REGION Network 10: J no magnet pallet ///Empty pallet full
   RUNG wire#powerrail
      Contact( "AlwaysTRUE" )
      Contact( "Station_Sys".Auto.Mode )
      wire#w1
      I_Contact( "AutoProcessControl".J_MagnetLine.Robot2PickPrimit )
      I_Contact( "iJ-magnetLiftingPalletDischargeDetection" )
      Coil( "ST10_TipDB".Global."6"[4] )
   END_RUNG
   RUNG wire#w1
      Contact( "iJ-magnetTakeShaftDetection" )
      { S7_Templates := "time_type := Time" } "TON".TON[48].TON(pt := T#3S, et =>)
      Coil( "ST10_TipDB".Global."6"[5] )
   END_RUNG
   // the same network as SCL:
   #_w1 := "AlwaysTRUE" AND "Station_Sys".Auto.Mode;
   "ST10_TipDB".Global."6"[4] := #_w1 AND NOT "AutoProcessControl".J_MagnetLine.Robot2PickPrimit AND NOT "iJ-magnetLiftingPalletDischargeDetection";
   "TON".TON[48].TON(IN := #_w1 AND "iJ-magnetTakeShaftDetection", PT := T#3S);
   "ST10_TipDB".Global."6"[5] := "TON".TON[48].Q;
END_REGION

REGION Network 11: K no magnet pallet ///Empty pallet full
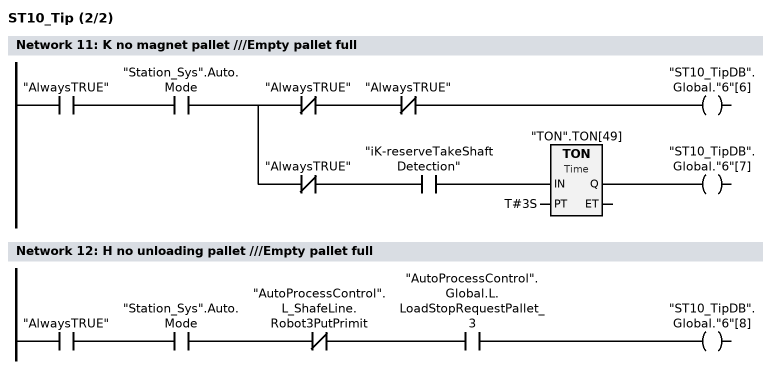
   RUNG wire#powerrail
      Contact( "AlwaysTRUE" )
      Contact( "Station_Sys".Auto.Mode )
      wire#w1
      I_Contact( "AlwaysTRUE" )
      I_Contact( "AlwaysTRUE" )
      Coil( "ST10_TipDB".Global."6"[6] )
   END_RUNG
   RUNG wire#w1
      I_Contact( "AlwaysTRUE" )
      Contact( "iK-reserveTakeShaftDetection" )
      { S7_Templates := "time_type := Time" } "TON".TON[49].TON(pt := T#3S, et =>)
      Coil( "ST10_TipDB".Global."6"[7] )
   END_RUNG
   // the same network as SCL:
   #_w1 := "AlwaysTRUE" AND "Station_Sys".Auto.Mode;
   "ST10_TipDB".Global."6"[6] := #_w1 AND NOT "AlwaysTRUE" AND NOT "AlwaysTRUE";
   "TON".TON[49].TON(IN := #_w1 AND NOT "AlwaysTRUE" AND "iK-reserveTakeShaftDetection", PT := T#3S);
   "ST10_TipDB".Global."6"[7] := "TON".TON[49].Q;
END_REGION

REGION Network 12: H no unloading pallet ///Empty pallet full
   RUNG wire#powerrail
      Contact( "AlwaysTRUE" )
      Contact( "Station_Sys".Auto.Mode )
      I_Contact( "AutoProcessControl".L_ShafeLine.Robot3PutPrimit )
      Contact( "AutoProcessControl".Global.L.LoadStopRequestPallet_3 )
      Coil( "ST10_TipDB".Global."6"[8] )
   END_RUNG
   // the same network as SCL:
   "ST10_TipDB".Global."6"[8] := "AlwaysTRUE" AND "Station_Sys".Auto.Mode AND NOT "AutoProcessControl".L_ShafeLine.Robot3PutPrimit AND "AutoProcessControl".Global.L.LoadStopRequestPallet_3;
END_REGION
END_FUNCTION

FUNCTION "CylinderCtrl_V2" : Void   // FC3011, SCL
TITLE = CylinderV3
{ S7_Optimized_Access := 'FALSE' }
AUTHOR : JM
FAMILY : RCS
VERSION : 18.2
// this function is only used for cylinder control
// stored: AutoNumber false, SetENOAutomatically true
   VAR_INPUT
      iReset : Bool;   // reset action
      iRun : Bool;   // system run
      iEStop : Bool;   // e_stop monitor
      iManualMode : Bool;   // manual mode
      iAutoMode : Bool;   // auto mode
      iEnableAlarm : Bool;   // alarm will popup up
      iPulse100mS : Bool;   // pulse *100ms
      iPulse1S : Bool;   // pulse*1s
      iCyDBNO : Word;   // Interface data block number
      iCyCounts : Int;   // total counts of cylinder to be used[must be>=1 and <=100]
      iDevAlarmDBNum : Word;   // Device Alarm DataBlock Alarm
   END_VAR
   VAR_TEMP
      CyInterface : "Cyl";
      CyRany : Any;
      cyRSany AT CyRany : Struct
         SyntaxID : Byte;
         DataType : Byte;
         RepetitionFactor : Int;
         DB_Number : Word;
         MemoryAreaAddress : DWord;
      END_STRUCT;
      CyDany : Any;
      CyDSany AT CyDany : Struct
         SyntaxID : Byte;
         DataType : Byte;
         RepetitionFactor : Int;
         DB_Number : Word;
         MemoryAreaAddress : DWord;
      END_STRUCT;
      tpCounts : Int;
      tpi : Int;
      tpRetVal : Int;
   END_VAR
BEGIN
   //---------------------------------------------------------------//
   //FunctionName:CylinderV3
   //FunctionDescription:Cylinder Control block
   //---------------------------------------------------------------//
   (*in:

   #iReset  Bool            reset action
   #iRun    Bool            system run
   #iE_stop Bool            e_stop monitor
   #iManualMode Bool        manual mode
   #iAutoMode   Bool        auto mode
   #iEnableAlarm    Bool        alarm will popup up
   #iPulse_100mS    Bool        pulse *100ms
   iPulse_1S   Bool        pulse*1s
   iCyDBNO Int Int     Interface data block number
   iCyCounts   Int     total counts OF "Cylinder" TO be used[must be>=1 AND <=100]

   //inout:
   //out:
   *)
   //---------------------------------------------------------------//
   //Version:V3
   //D&T:2016-11-14
   //Group:RCS
   //Author:JiangMing
   //-------------------------Modify1----------------------------------//
   //Version:
   //D&T:2016-11-17
   //Group: RCS
   //Author:JiangMing
   //Modify:Update cylinder no as output interface
   //-------------------------Modify2----------------------------------//
   //Version:       V18.3
   //D&T:           2020-06-11
   //Group:         RCS
   //Author:        JM
   //Modify:        1.MaxCylinder count 200 
   //               2.Refine alarm interface
   IF #iCyCounts > 200 THEN
       #tpCounts := 200;
   ELSE
       #tpCounts := #iCyCounts;
   END_IF;
   //input

   FOR #tpi := 0 TO #tpCounts-1 DO
       //****************************************************************************************//
       #cyRSany.SyntaxID := 16#10;
       #cyRSany.DataType := 16#02;
       #cyRSany.RepetitionFactor := 22;
       #cyRSany.DB_Number := #iCyDBNO;
       #cyRSany.MemoryAreaAddress := 16#8400_0000 OR (SHL(IN := INT_TO_DWORD(#tpi * 22), N := 3));///
       //-----------------------------//
       #CyDSany.SyntaxID := 16#10;
       #CyDSany.DataType := 16#02;
       #CyDSany.RepetitionFactor := 22;
       #CyDSany.DB_Number := 0;
       #CyDSany.MemoryAreaAddress := 16#8700_0000 OR (SHL(IN := INT_TO_DWORD(0), N := 3));///
       #tpRetVal := BLKMOV(SRCBLK := #CyRany, DSTBLK => #CyDany);
       //***************************************************************************************//
       "CylinderModule_V2"(iReset := #iReset,
                        iRun := #iRun,
                        iEStop := #iEStop,
                        iManualMode := #iManualMode,
                        iAutoMode := #iAutoMode,
                        iEnableAlarm := #iEnableAlarm,
                        iPulse100mS := #iPulse100mS,
                        iPulse1S := #iPulse1S,
                        iError := #CyInterface.In.Error,
                        iGoWorkInterlock := #CyInterface.In.GoWorkInterlock,
                        iGoHomeInterlock := #CyInterface.In.GoHomeInterlock,
                        iWorkPositionSensor := #CyInterface.In.WorkPositionSensor,
                        iHomePositionSensor := #CyInterface.In.HomePositionSensor,
                        iValveType := #CyInterface.In.ValveType,
                        iManualOutputType := #CyInterface.In.ManualOutputType,
                        iFaultTime := #CyInterface.In.FaultTime,
                        iOnPositionTime := #CyInterface.In.OnPositionTime,
                           ioResetOut:=#CyInterface.Inout.ResetOut,
                        ioGoWorkPosition := #CyInterface.Out.GoWorkPosition,
                        ioGoHomePosition := #CyInterface.Out.GoHomePosition,
                        oGoWP_ButtonActive => #CyInterface.Out.GoWPButtonActive,
                        oGoHP_ButtonActive => #CyInterface.Out.GoHPButtonActive,
                        ioGoWorkFault := #CyInterface.Out.GoWorkFault,
                        ioGoHomeFault := #CyInterface.Out.GoHomeFault,
                        ioSensorPositionFault := #CyInterface.Out.SensorPositionFault,
                        oCyNo => #CyInterface.Out.CyNO,
                        ioManualGoWork := #CyInterface.Inout.ManualGoWork,
                        ioManualGoHome := #CyInterface.Inout.ManualGoHome,
                        ioAutoGoWork := #CyInterface.Inout.AutoGoWork,
                        ioAutoGoHome := #CyInterface.Inout.AutoGoHome,
                        ioGoWorkTime := #CyInterface.S.GoWorkTime,
                        ioGoHomeTime := #CyInterface.S.GoHomeTime,
                        ioWorkFaultTime := #CyInterface.S.WorkFaultTime,
                        ioHomeFaultTime := #CyInterface.S.HomeFaultTime,
                        ioBothSensorOnTime := #CyInterface.S.BothSensorOnTime,
                        ioPulse100mSP := #CyInterface.S.Pulse100mSP,
                        ioAutoGoWorkP := #CyInterface.S.AutoGoWorkP,
                        ioAutoGoHomeP := #CyInterface.S.AutoGoHomeP,
                        ioGoWork100mSP := #CyInterface.S.GoWork100mSP,
                        ioGoHome100mSP := #CyInterface.S.GoHome100mSP,
                        ioBothSensorOn100mSP := #CyInterface.S.BothSensorOn100mSP,
                        ioAlarm := #CyInterface.S.Alarm,
                        ioSpare1 := #CyInterface.S.spare1,
                        ioSpare2 := #CyInterface.S.spare2);
       //*******************************************************************************//
         POKE_BOOL(area := 16#84,
                   bitOffset := 4 * (#tpi MOD 2) + 0,
                   byteOffset :=  #tpi / 2,
                   dbNumber := #iDevAlarmDBNum,
                   value := #CyInterface.Out.GoWorkFault);
         POKE_BOOL(area := 16#84,
                   bitOffset := 4 * (#tpi MOD 2) + 1,
                   byteOffset :=  #tpi / 2,
                   dbNumber := #iDevAlarmDBNum,
                   value := #CyInterface.Out.GoHomeFault);
         POKE_BOOL(area := 16#84,
                   bitOffset := 4 * (#tpi MOD 2) + 2,
                   byteOffset :=  #tpi / 2,
                   dbNumber := #iDevAlarmDBNum,
                   value := #CyInterface.Out.SensorPositionFault);
       #CyInterface.Out.CyNO := INT_TO_BYTE(#tpi+1);
       //output
       #cyRSany.SyntaxID := 16#10;
       #cyRSany.DataType := 16#02;
       #cyRSany.RepetitionFactor := 16;
       #cyRSany.DB_Number := 0;
       #cyRSany.MemoryAreaAddress := 16#8700_0000 OR (SHL(IN := INT_TO_DWORD(6), N := 3));///
       //-----------------------------//
       #CyDSany.SyntaxID := 16#10;
       #CyDSany.DataType := 16#02;
       #CyDSany.RepetitionFactor := 16;
       #CyDSany.DB_Number := #iCyDBNO;
       #CyDSany.MemoryAreaAddress := 16#8400_0000 OR (SHL(IN := INT_TO_DWORD(#tpi* 22 + 6), N := 3));///
       #tpRetVal := BLKMOV(SRCBLK := #CyRany, DSTBLK => #CyDany);
       //******************************************************************************//


   END_FOR;
END_FUNCTION

FUNCTION "ST10Cyl_interface1-10" : Void   // FC1020, LAD
{ S7_Optimized_Access := 'FALSE' }
// stored: AutoNumber false, SetENOAutomatically false
   VAR_INPUT
      AlwaysON : Bool;
      E_stop : Bool;
   END_VAR
   VAR_TEMP
      tTest : Bool;
      i : Int;
   END_VAR
BEGIN

REGION Network 1 (SCL): Cylinder 1-10 IO Interface (SCL)
   IF "Station_Sys".Manual.Mode THEN

       FOR #i := 1 TO 100 BY 1

       DO
           "ST10Cylinder".Cy[#i].In.ManualOutputType := TRUE;

       END_FOR;

   END_IF;

   //Cylinder1 IO  A-Loading-01HorizontalCylinder
   //Input
   "ST10Cylinder".Cy[1].In.WorkPositionSensor := "iA-Loading-01HorizontalCylinderInWP";
   "ST10Cylinder".Cy[1].In.HomePositionSensor := "iA-Loading-01HorizontalCylinderInHP";
   //Output
   "oA-Loading-01HorizontalCylinderToWP" := "ST10Cylinder".Cy[1].Out.GoWorkPosition;
   "oA-Loading-01HorizontalCylinderToHP" := "ST10Cylinder".Cy[1].Out.GoHomePosition;

   //Cylinder2 IO  A-Loading-01UpDownTakeCylinder
   //Input
   "ST10Cylinder".Cy[2].In.WorkPositionSensor := "iA-Loading-01UpDownTakeCylinderInWP";
   "ST10Cylinder".Cy[2].In.HomePositionSensor := "iA-Loading-01UpDownTakeCylinderInHP";
   //Output
   "oA-Loading-01UpDownTakeCylinderToWP" := "ST10Cylinder".Cy[2].Out.GoWorkPosition;
   "oA-Loading-01UpDownTakeCylinderToHP" := "ST10Cylinder".Cy[2].Out.GoHomePosition;

   //Cylinder3 IO  A-Loading-02HorizontalCylinder
   //Input
   "ST10Cylinder".Cy[3].In.WorkPositionSensor := "iA-Loading-02HorizontalCylinderInWP"  ;
   "ST10Cylinder".Cy[3].In.HomePositionSensor := "iA-Loading-02HorizontalCylinderInHP"  ;
   //Output
   "oA-Loading-02HorizontalCylinderToWP" := "ST10Cylinder".Cy[3].Out.GoWorkPosition;
   "oA-Loading-02HorizontalCylinderToHP" := "ST10Cylinder".Cy[3].Out.GoHomePosition;

   //Cylinder4 IO     A-Loading-02UpDownTakeCylinder
   //Input
   "ST10Cylinder".Cy[4].In.WorkPositionSensor := "iA-Loading-02UpDownTakeCylinderInWP";
   "ST10Cylinder".Cy[4].In.HomePositionSensor := "iA-Loading-02UpDownTakeCylinderInHP";
   //Output
   "oA-Loading-02UpDownTakeCylinderToWP" := "ST10Cylinder".Cy[4].Out.GoWorkPosition;
   "oA-Loading-02UpDownTakeCylinderToHP" := "ST10Cylinder".Cy[4].Out.GoHomePosition;

   //Cylinder5 IO  B-PressFitting-01GripperCylinder
   //Input
   "ST10Cylinder".Cy[5].In.WorkPositionSensor := "iB-PressFitting-01GripperCylinderInWP";
   "ST10Cylinder".Cy[5].In.HomePositionSensor := "iB-PressFitting-01GripperCylinderInHP";
   //Output
   "oB-PressFitting-01GripperCylinderToWP" := "ST10Cylinder".Cy[5].Out.GoWorkPosition;
   "oB-PressFitting-01GripperCylinderToHP" := "ST10Cylinder".Cy[5].Out.GoHomePosition;

   //Cylinder6 IO  B-PressFitting-01Cylinder
   //Input
   "ST10Cylinder".Cy[6].In.WorkPositionSensor := "iB-PressFitting-01CylinderInWP" ;
   "ST10Cylinder".Cy[6].In.HomePositionSensor := "iB-PressFitting-01CylinderInHP" ;
   //Output
   "oB-PressFitting-01CylinderToWP" := "ST10Cylinder".Cy[6].Out.GoWorkPosition;
   "oB-PressFitting-01CylinderToHP" := "ST10Cylinder".Cy[6].Out.GoHomePosition;

   //Cylinder7 IO  B-PressFitting-02GripperCylinder
   //Input
   "ST10Cylinder".Cy[7].In.WorkPositionSensor := "iB-PressFitting-02GripperCylinderInWP";
   "ST10Cylinder".Cy[7].In.HomePositionSensor := "iB-PressFitting-02GripperCylinderInHP";
   //Output
   "oB-PressFitting-02GripperCylinderToWP" := "ST10Cylinder".Cy[7].Out.GoWorkPosition;
   "oB-PressFitting-02GripperCylinderToHP" := "ST10Cylinder".Cy[7].Out.GoHomePosition;

   //Cylinder8 IO  B-PressFitting-02Cylinder
   //Input
   "ST10Cylinder".Cy[8].In.WorkPositionSensor := "iB-PressFitting-02CylinderInWP";
   "ST10Cylinder".Cy[8].In.HomePositionSensor := "iB-PressFitting-02CylinderInHP";
   //Output
   "oB-PressFitting-02CylinderToWP" := "ST10Cylinder".Cy[8].Out.GoWorkPosition;
   "oB-PressFitting-02CylinderToHP" := "ST10Cylinder".Cy[8].Out.GoHomePosition;

   //Cylinder9 IO  C-LocationCylinder
   //Input
   "ST10Cylinder".Cy[9].In.WorkPositionSensor := "iC-LocationCylinderInWP";
   "ST10Cylinder".Cy[9].In.HomePositionSensor := "iC-LocationCylinderInHP";
   //Output
   "oC-LocationCylinderToWP" := "ST10Cylinder".Cy[9].Out.GoWorkPosition;
   "oC-LocationCylinderToHP" := "ST10Cylinder".Cy[9].Out.GoHomePosition;


   //Cylinder10 IO  Spare
   //Input
   "ST10Cylinder".Cy[10].In.WorkPositionSensor := "ST10Cylinder".Cy[10].Out.GoWorkPosition ;
   "ST10Cylinder".Cy[10].In.HomePositionSensor := "ST10Cylinder".Cy[10].Out.GoHomePosition ;
   //Output
   "ST10Cylinder".Cy[10].Out.GoWorkPosition := "ST10Cylinder".Cy[10].Out.GoWorkPosition;
   "ST10Cylinder".Cy[10].Out.GoHomePosition := "ST10Cylinder".Cy[10].Out.GoHomePosition;
END_REGION

REGION Network 2: CY1 interface A-Loading-01HorizontalCylinder
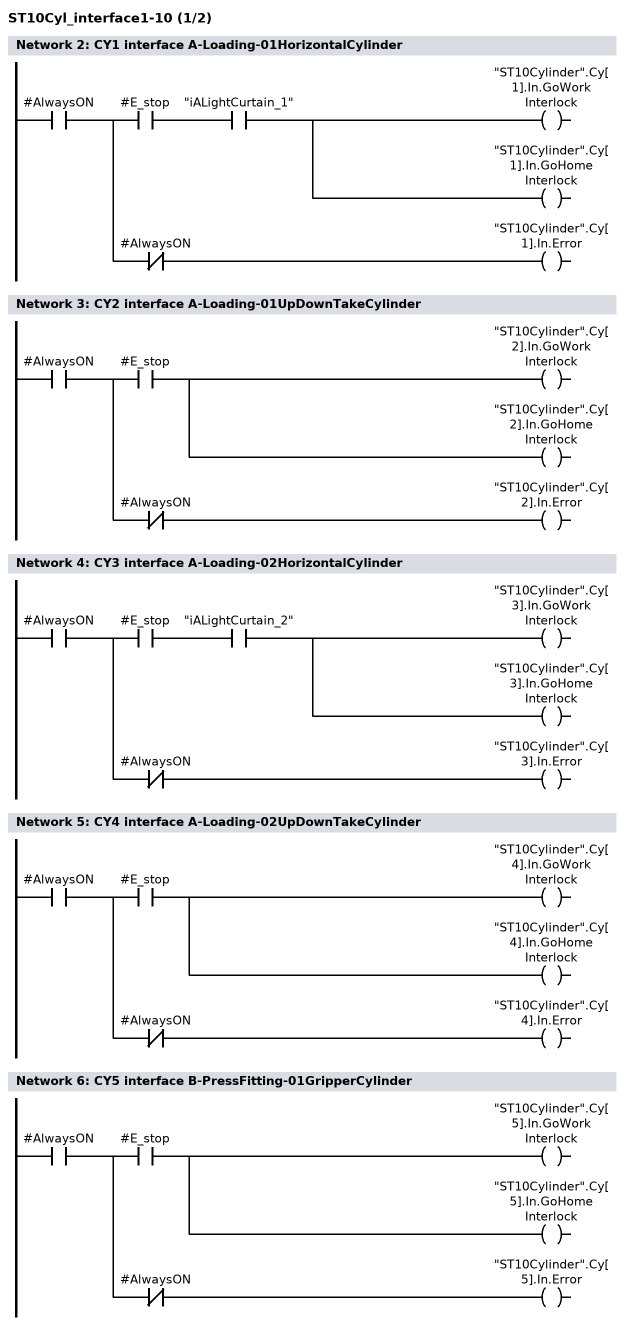
   RUNG wire#powerrail
      Contact( #AlwaysON )
      wire#w1
      Contact( #E_stop )
      Contact( "iALightCurtain_1" )
      wire#w2
      Coil( "ST10Cylinder".Cy[1].In.GoWorkInterlock )
   END_RUNG
   RUNG wire#w2
      Coil( "ST10Cylinder".Cy[1].In.GoHomeInterlock )
   END_RUNG
   RUNG wire#w1
      I_Contact( #AlwaysON )
      Coil( "ST10Cylinder".Cy[1].In.Error )
   END_RUNG
   // the same network as SCL:
   "ST10Cylinder".Cy[1].In.GoWorkInterlock := #AlwaysON AND #E_stop AND "iALightCurtain_1";
   "ST10Cylinder".Cy[1].In.GoHomeInterlock := #AlwaysON AND #E_stop AND "iALightCurtain_1";
   "ST10Cylinder".Cy[1].In.Error := #AlwaysON AND NOT #AlwaysON;
END_REGION

REGION Network 3: CY2 interface A-Loading-01UpDownTakeCylinder
   RUNG wire#powerrail
      Contact( #AlwaysON )
      wire#w1
      Contact( #E_stop )
      wire#w2
      Coil( "ST10Cylinder".Cy[2].In.GoWorkInterlock )
   END_RUNG
   RUNG wire#w2
      Coil( "ST10Cylinder".Cy[2].In.GoHomeInterlock )
   END_RUNG
   RUNG wire#w1
      I_Contact( #AlwaysON )
      Coil( "ST10Cylinder".Cy[2].In.Error )
   END_RUNG
   // the same network as SCL:
   "ST10Cylinder".Cy[2].In.GoWorkInterlock := #AlwaysON AND #E_stop;
   "ST10Cylinder".Cy[2].In.GoHomeInterlock := #AlwaysON AND #E_stop;
   "ST10Cylinder".Cy[2].In.Error := #AlwaysON AND NOT #AlwaysON;
END_REGION

REGION Network 4: CY3 interface A-Loading-02HorizontalCylinder
   RUNG wire#powerrail
      Contact( #AlwaysON )
      wire#w1
      Contact( #E_stop )
      Contact( "iALightCurtain_2" )
      wire#w2
      Coil( "ST10Cylinder".Cy[3].In.GoWorkInterlock )
   END_RUNG
   RUNG wire#w2
      Coil( "ST10Cylinder".Cy[3].In.GoHomeInterlock )
   END_RUNG
   RUNG wire#w1
      I_Contact( #AlwaysON )
      Coil( "ST10Cylinder".Cy[3].In.Error )
   END_RUNG
   // the same network as SCL:
   "ST10Cylinder".Cy[3].In.GoWorkInterlock := #AlwaysON AND #E_stop AND "iALightCurtain_2";
   "ST10Cylinder".Cy[3].In.GoHomeInterlock := #AlwaysON AND #E_stop AND "iALightCurtain_2";
   "ST10Cylinder".Cy[3].In.Error := #AlwaysON AND NOT #AlwaysON;
END_REGION

REGION Network 5: CY4 interface A-Loading-02UpDownTakeCylinder
   RUNG wire#powerrail
      Contact( #AlwaysON )
      wire#w1
      Contact( #E_stop )
      wire#w2
      Coil( "ST10Cylinder".Cy[4].In.GoWorkInterlock )
   END_RUNG
   RUNG wire#w2
      Coil( "ST10Cylinder".Cy[4].In.GoHomeInterlock )
   END_RUNG
   RUNG wire#w1
      I_Contact( #AlwaysON )
      Coil( "ST10Cylinder".Cy[4].In.Error )
   END_RUNG
   // the same network as SCL:
   "ST10Cylinder".Cy[4].In.GoWorkInterlock := #AlwaysON AND #E_stop;
   "ST10Cylinder".Cy[4].In.GoHomeInterlock := #AlwaysON AND #E_stop;
   "ST10Cylinder".Cy[4].In.Error := #AlwaysON AND NOT #AlwaysON;
END_REGION

REGION Network 6: CY5 interface B-PressFitting-01GripperCylinder
   RUNG wire#powerrail
      Contact( #AlwaysON )
      wire#w1
      Contact( #E_stop )
      wire#w2
      Coil( "ST10Cylinder".Cy[5].In.GoWorkInterlock )
   END_RUNG
   RUNG wire#w2
      Coil( "ST10Cylinder".Cy[5].In.GoHomeInterlock )
   END_RUNG
   RUNG wire#w1
      I_Contact( #AlwaysON )
      Coil( "ST10Cylinder".Cy[5].In.Error )
   END_RUNG
   // the same network as SCL:
   "ST10Cylinder".Cy[5].In.GoWorkInterlock := #AlwaysON AND #E_stop;
   "ST10Cylinder".Cy[5].In.GoHomeInterlock := #AlwaysON AND #E_stop;
   "ST10Cylinder".Cy[5].In.Error := #AlwaysON AND NOT #AlwaysON;
END_REGION

REGION Network 7: CY6 interface B-PressFitting-01Cylinder
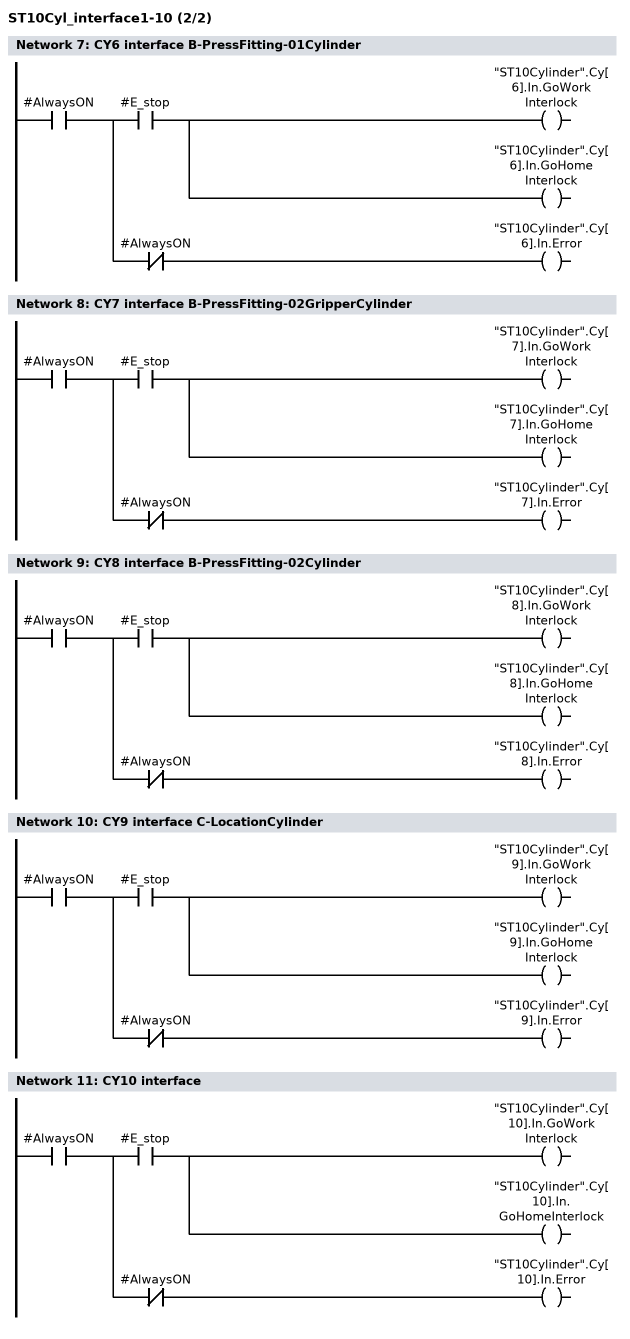
   RUNG wire#powerrail
      Contact( #AlwaysON )
      wire#w1
      Contact( #E_stop )
      wire#w2
      Coil( "ST10Cylinder".Cy[6].In.GoWorkInterlock )
   END_RUNG
   RUNG wire#w2
      Coil( "ST10Cylinder".Cy[6].In.GoHomeInterlock )
   END_RUNG
   RUNG wire#w1
      I_Contact( #AlwaysON )
      Coil( "ST10Cylinder".Cy[6].In.Error )
   END_RUNG
   // the same network as SCL:
   "ST10Cylinder".Cy[6].In.GoWorkInterlock := #AlwaysON AND #E_stop;
   "ST10Cylinder".Cy[6].In.GoHomeInterlock := #AlwaysON AND #E_stop;
   "ST10Cylinder".Cy[6].In.Error := #AlwaysON AND NOT #AlwaysON;
END_REGION

REGION Network 8: CY7 interface B-PressFitting-02GripperCylinder
   RUNG wire#powerrail
      Contact( #AlwaysON )
      wire#w1
      Contact( #E_stop )
      wire#w2
      Coil( "ST10Cylinder".Cy[7].In.GoWorkInterlock )
   END_RUNG
   RUNG wire#w2
      Coil( "ST10Cylinder".Cy[7].In.GoHomeInterlock )
   END_RUNG
   RUNG wire#w1
      I_Contact( #AlwaysON )
      Coil( "ST10Cylinder".Cy[7].In.Error )
   END_RUNG
   // the same network as SCL:
   "ST10Cylinder".Cy[7].In.GoWorkInterlock := #AlwaysON AND #E_stop;
   "ST10Cylinder".Cy[7].In.GoHomeInterlock := #AlwaysON AND #E_stop;
   "ST10Cylinder".Cy[7].In.Error := #AlwaysON AND NOT #AlwaysON;
END_REGION

REGION Network 9: CY8 interface B-PressFitting-02Cylinder
   RUNG wire#powerrail
      Contact( #AlwaysON )
      wire#w1
      Contact( #E_stop )
      wire#w2
      Coil( "ST10Cylinder".Cy[8].In.GoWorkInterlock )
   END_RUNG
   RUNG wire#w2
      Coil( "ST10Cylinder".Cy[8].In.GoHomeInterlock )
   END_RUNG
   RUNG wire#w1
      I_Contact( #AlwaysON )
      Coil( "ST10Cylinder".Cy[8].In.Error )
   END_RUNG
   // the same network as SCL:
   "ST10Cylinder".Cy[8].In.GoWorkInterlock := #AlwaysON AND #E_stop;
   "ST10Cylinder".Cy[8].In.GoHomeInterlock := #AlwaysON AND #E_stop;
   "ST10Cylinder".Cy[8].In.Error := #AlwaysON AND NOT #AlwaysON;
END_REGION

REGION Network 10: CY9 interface C-LocationCylinder
   RUNG wire#powerrail
      Contact( #AlwaysON )
      wire#w1
      Contact( #E_stop )
      wire#w2
      Coil( "ST10Cylinder".Cy[9].In.GoWorkInterlock )
   END_RUNG
   RUNG wire#w2
      Coil( "ST10Cylinder".Cy[9].In.GoHomeInterlock )
   END_RUNG
   RUNG wire#w1
      I_Contact( #AlwaysON )
      Coil( "ST10Cylinder".Cy[9].In.Error )
   END_RUNG
   // the same network as SCL:
   "ST10Cylinder".Cy[9].In.GoWorkInterlock := #AlwaysON AND #E_stop;
   "ST10Cylinder".Cy[9].In.GoHomeInterlock := #AlwaysON AND #E_stop;
   "ST10Cylinder".Cy[9].In.Error := #AlwaysON AND NOT #AlwaysON;
END_REGION

REGION Network 11: CY10 interface
   RUNG wire#powerrail
      Contact( #AlwaysON )
      wire#w1
      Contact( #E_stop )
      wire#w2
      Coil( "ST10Cylinder".Cy[10].In.GoWorkInterlock )
   END_RUNG
   RUNG wire#w2
      Coil( "ST10Cylinder".Cy[10].In.GoHomeInterlock )
   END_RUNG
   RUNG wire#w1
      I_Contact( #AlwaysON )
      Coil( "ST10Cylinder".Cy[10].In.Error )
   END_RUNG
   // the same network as SCL:
   "ST10Cylinder".Cy[10].In.GoWorkInterlock := #AlwaysON AND #E_stop;
   "ST10Cylinder".Cy[10].In.GoHomeInterlock := #AlwaysON AND #E_stop;
   "ST10Cylinder".Cy[10].In.Error := #AlwaysON AND NOT #AlwaysON;
END_REGION
END_FUNCTION

FUNCTION "ST10Cyl_interface11-20" : Void   // FC1021, LAD
{ S7_Optimized_Access := 'FALSE' }
// stored: AutoNumber false, SetENOAutomatically false
   VAR_INPUT
      AlwaysON : Bool;
      E_stop : Bool;
   END_VAR
   VAR_TEMP
      tTest : Bool;
   END_VAR
BEGIN

REGION Network 1 (SCL): Cylinder 11-20 IO Interface (SCL)

   //Cylinder11 IO   E-NG-01NGLocationCylinder
   //Input
   "ST10Cylinder".Cy[11].In.WorkPositionSensor := "iE-NG-01NGLocationCylinderInWP";
   "ST10Cylinder".Cy[11].In.HomePositionSensor := "iE-NG-01NGLocationCylinderInHP";
   //Output
   "oE-NG-01NGLocationCylinderToWP" := "ST10Cylinder".Cy[11].Out.GoWorkPosition;
   "oE-NG-01NGLocationCylinderToHP" := "ST10Cylinder".Cy[11].Out.GoHomePosition;

   //Cylinder12 IO  E-NG-02NGLocationCylinder
   //Input
   "ST10Cylinder".Cy[12].In.WorkPositionSensor := "iE-NG-02NGLocationCylinderInWP";
   "ST10Cylinder".Cy[12].In.HomePositionSensor := "iE-NG-02NGLocationCylinderInHP";
   //Output
   "oE-NG-02NGLocationCylinderToWP" := "ST10Cylinder".Cy[12].Out.GoWorkPosition;
   "oE-NG-02NGLocationCylinderToHP" := "ST10Cylinder".Cy[12].Out.GoHomePosition;

   //Cylinder13 IO  F-ROOBT1Gripper1Cylinder
   //Input
   "KukaRobot1_CtrlDB".sPLCtoROB.User.Gripper.DI129_Grip1WP:="ST10Cylinder".Cy[13].In.WorkPositionSensor := "iF-ROOBT1Gripper1CylinderInWP" ;
   "KukaRobot1_CtrlDB".sPLCtoROB.User.Gripper.DI130_Grip1HP := "ST10Cylinder".Cy[13].In.HomePositionSensor := "iF-ROOBT1Gripper1CylinderInHP" ;//"TON".TON[0].Q;

   IF  NOT "Robot_DB".Control.Robot1GripControl THEN
       //Output
       "oF-ROOBT1Gripper1CylinderToWP" := "KukaRobot1_CtrlDB".sROBtoPLC.User.Gripper.DO129_Grip1GoWork;
       "oF-ROOBT1Gripper1CylinderToHP" := "KukaRobot1_CtrlDB".sROBtoPLC.User.Gripper.DO130_Grip1GoHome;
   ELSE
       //Output
       "oF-ROOBT1Gripper1CylinderToWP" := "ST10Cylinder".Cy[13].Out.GoWorkPosition;
       "oF-ROOBT1Gripper1CylinderToHP" := "ST10Cylinder".Cy[13].Out.GoHomePosition;
   END_IF;
   "TON".TON[0](IN:="oF-ROOBT1Gripper1CylinderToHP" AND NOT"iF-ROOBT1Gripper1CylinderInWP",PT:=T#500MS);


   //Cylinder14 IO  F-ROOBT1Gripper2Cylinder
   //Input
   "KukaRobot1_CtrlDB".sPLCtoROB.User.Gripper.DI131_Grip2WP:="ST10Cylinder".Cy[14].In.WorkPositionSensor := "iF-ROOBT1Gripper2CylinderInWP";
   "KukaRobot1_CtrlDB".sPLCtoROB.User.Gripper.DI132_Grip2HP:="ST10Cylinder".Cy[14].In.HomePositionSensor := "iF-ROOBT1Gripper2CylinderInHP";

   IF NOT "Robot_DB".Control.Robot1GripControl THEN
       //Output
       "oF-ROOBT1Gripper2CylinderToWP" :="ST10Cylinder".Cy[14].Inout.AutoGoWork:="KukaRobot1_CtrlDB".sROBtoPLC.User.Gripper.DO131_Grip2GoWork;
       "oF-ROOBT1Gripper2CylinderToHP" :="ST10Cylinder".Cy[14].Inout.AutoGoHome:="KukaRobot1_CtrlDB".sROBtoPLC.User.Gripper.DO132_Grip2GoHome;
   ELSE
       //Output
       "oF-ROOBT1Gripper2CylinderToWP" := "ST10Cylinder".Cy[14].Out.GoWorkPosition;
       "oF-ROOBT1Gripper2CylinderToHP" := "ST10Cylinder".Cy[14].Out.GoHomePosition;
   END_IF;


   //Cylinder15 IO  F-ROOBT2Gripper1Cylinder
   //Input
   "KukaRobot2_CtrlDB".sPLCtoROB.User.Gripper.DI129_Grip1WP:="ST10Cylinder".Cy[15].In.WorkPositionSensor := "iF-ROOBT2Gripper1CylinderInWP";
   "KukaRobot2_CtrlDB".sPLCtoROB.User.Gripper.DI130_Grip1HP := "ST10Cylinder".Cy[15].In.HomePositionSensor :="iF-ROOBT2Gripper1CylinderInHP";

   IF NOT "Robot_DB".Control.Robot2GripControl THEN
       //Output
       "oF-ROOBT2Gripper1CylinderToWP" :="ST10Cylinder".Cy[15].Inout.AutoGoWork:="KukaRobot2_CtrlDB".sROBtoPLC.User.Gripper.DO129_Grip1GoWork;
       "oF-ROOBT2Gripper1CylinderToHP" :="ST10Cylinder".Cy[15].Inout.AutoGoHome:="KukaRobot2_CtrlDB".sROBtoPLC.User.Gripper.DO130_Grip1GoHome;
   ELSE
       //Output
       "oF-ROOBT2Gripper1CylinderToWP" := "ST10Cylinder".Cy[15].Out.GoWorkPosition;
       "oF-ROOBT2Gripper1CylinderToHP" := "ST10Cylinder".Cy[15].Out.GoHomePosition;
   END_IF;



   //Cylinder16 IO  F-ROOBT2Gripper2Cylinder
   //Input
   "KukaRobot2_CtrlDB".sPLCtoROB.User.Gripper.DI131_Grip2WP:="ST10Cylinder".Cy[16].In.WorkPositionSensor := "iF-ROOBT2Gripper2CylinderInWP";
   "KukaRobot2_CtrlDB".sPLCtoROB.User.Gripper.DI132_Grip2HP:="ST10Cylinder".Cy[16].In.HomePositionSensor := "iF-ROOBT2Gripper2CylinderInHP";

   IF NOT "Robot_DB".Control.Robot2GripControl THEN
       //Output
       "oF-ROOBT2Gripper2CylinderToWP" :="ST10Cylinder".Cy[16].Inout.AutoGoWork:= "KukaRobot2_CtrlDB".sROBtoPLC.User.Gripper.DO131_Grip2GoWork;
       "oF-ROOBT2Gripper2CylinderToHP" :="ST10Cylinder".Cy[16].Inout.AutoGoHome:= "KukaRobot2_CtrlDB".sROBtoPLC.User.Gripper.DO132_Grip2GoHome;
   ELSE
       //Output
       "oF-ROOBT2Gripper2CylinderToWP" := "ST10Cylinder".Cy[16].Out.GoWorkPosition;
       "oF-ROOBT2Gripper2CylinderToHP" := "ST10Cylinder".Cy[16].Out.GoHomePosition;
   END_IF;

   //Cylinder17 IO  F-ROOBT3Gripper1Cylinder
   //Input
   "KukaRobot3_CtrlDB".sPLCtoROB.User.Gripper.DI129_Grip1WP:="ST10Cylinder".Cy[17].In.WorkPositionSensor := "iF-ROOBT3Gripper1CylinderInWP";
   "KukaRobot3_CtrlDB".sPLCtoROB.User.Gripper.DI130_Grip1HP:="ST10Cylinder".Cy[17].In.HomePositionSensor := "iF-ROOBT3Gripper1CylinderInHP";

   IF NOT "Robot_DB".Control.Robot3GripControl THEN
       //Output
       "oF-ROOBT3Gripper1CylinderToWP" :="ST10Cylinder".Cy[17].Inout.AutoGoWork:="KukaRobot3_CtrlDB".sROBtoPLC.User.Gripper.DO129_Grip1GoWork;
       "oF-ROOBT3Gripper1CylinderToHP" :="ST10Cylinder".Cy[17].Inout.AutoGoHome:="KukaRobot3_CtrlDB".sROBtoPLC.User.Gripper.DO130_Grip1GoHome;
   ELSE
       //Output
       "oF-ROOBT3Gripper1CylinderToWP" := "ST10Cylinder".Cy[17].Out.GoWorkPosition;
       "oF-ROOBT3Gripper1CylinderToHP" := "ST10Cylinder".Cy[17].Out.GoHomePosition;
   END_IF;


   //Cylinder18 IO  F-ROOBT3Gripper2Cylinder
   //Input
   "KukaRobot3_CtrlDB".sPLCtoROB.User.Gripper.DI131_Grip2WP:="ST10Cylinder".Cy[18].In.WorkPositionSensor := "iF-ROOBT3Gripper2CylinderInWP";
   "KukaRobot3_CtrlDB".sPLCtoROB.User.Gripper.DI132_Grip2HP := "ST10Cylinder".Cy[18].In.HomePositionSensor := "iF-ROOBT3Gripper2CylinderInHP";//"TON".TON[1].Q;

   IF NOT "Robot_DB".Control.Robot3GripControl THEN
       //Output
       "oF-ROOBT3Gripper2CylinderToWP" :="ST10Cylinder".Cy[18].Inout.AutoGoWork:="KukaRobot3_CtrlDB".sROBtoPLC.User.Gripper.DO131_Grip2GoWork;
       "oF-ROOBT3Gripper2CylinderToHP" :="ST10Cylinder".Cy[18].Inout.AutoGoHome:="KukaRobot3_CtrlDB".sROBtoPLC.User.Gripper.DO132_Grip2GoHome;
   ELSE
       //Output
       "oF-ROOBT3Gripper2CylinderToWP" := "ST10Cylinder".Cy[18].Out.GoWorkPosition;
       "oF-ROOBT3Gripper2CylinderToHP" := "ST10Cylinder".Cy[18].Out.GoHomePosition;
   END_IF;

   "TON".TON[1](IN := "oF-ROOBT3Gripper2CylinderToHP" AND NOT "iF-ROOBT3Gripper2CylinderInWP",
                PT := T#500MS);

   (*
   //Cylinder19 IO  D-washer Loading Horizontal
   //Input
   "ST10Cylinder".Cy[19].In.WorkPositionSensor := ("D-washer Loading Cylinder Middle Cylinder InHP" AND "D-washer Loading Horizontal Cylinder InWP")
                                               OR ("D-washer Loading Cylinder Middle Cylinder InWP" AND "D-washer Loading Horizontal Cylinder InWP1");
   "ST10Cylinder".Cy[19].In.HomePositionSensor := "D-washer Loading Horizontal Cylinder InHP";
   //Output
   "D-washer Loading Horizontal Cylinder ToWP" := "ST10Cylinder".Cy[19].Out.GoWorkPosition;
   "D-washer Loading Horizontal Cylinder ToHP" := "ST10Cylinder".Cy[19].Out.GoHomePosition;

   //Cylinder20 IO  D-washer Loading Cylinder Middle
   //Input
   "ST10Cylinder".Cy[20].In.WorkPositionSensor := "D-washer Loading Cylinder Middle Cylinder InWP";
   "ST10Cylinder".Cy[20].In.HomePositionSensor := "D-washer Loading Cylinder Middle Cylinder InHP";
   //Output
   "D-washer Loading Cylinder Middle Cylinder ToWP" := "ST10Cylinder".Cy[20].Out.GoWorkPosition;
   "D-washer Loading Cylinder Middle Cylinder ToHP" := "ST10Cylinder".Cy[20].Out.GoHomePosition;
   *)
END_REGION

REGION Network 2: CY11 interface E-NG-01NGLocationCylinder
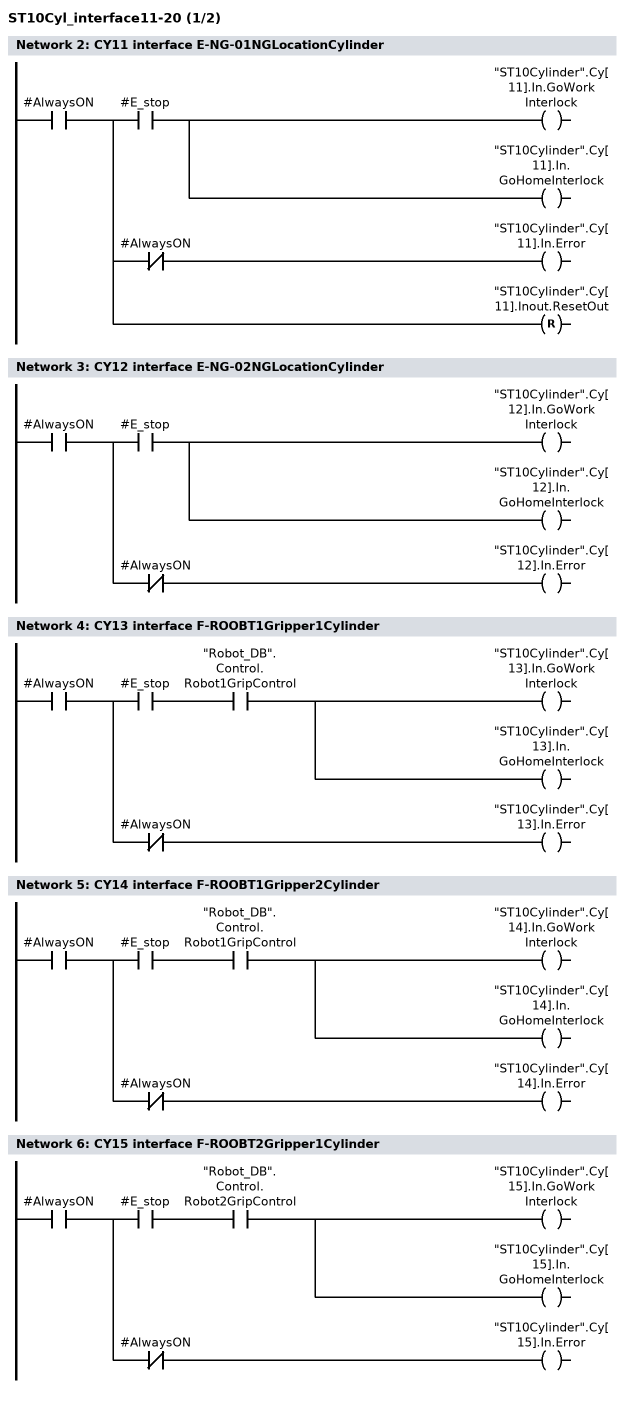
   RUNG wire#powerrail
      Contact( #AlwaysON )
      wire#w1
      Contact( #E_stop )
      wire#w2
      Coil( "ST10Cylinder".Cy[11].In.GoWorkInterlock )
   END_RUNG
   RUNG wire#w2
      Coil( "ST10Cylinder".Cy[11].In.GoHomeInterlock )
   END_RUNG
   RUNG wire#w1
      I_Contact( #AlwaysON )
      Coil( "ST10Cylinder".Cy[11].In.Error )
   END_RUNG
   RUNG wire#w1
      R_Coil( "ST10Cylinder".Cy[11].Inout.ResetOut )
   END_RUNG
   // the same network as SCL:
   "ST10Cylinder".Cy[11].In.GoWorkInterlock := #AlwaysON AND #E_stop;
   "ST10Cylinder".Cy[11].In.GoHomeInterlock := #AlwaysON AND #E_stop;
   "ST10Cylinder".Cy[11].In.Error := #AlwaysON AND NOT #AlwaysON;
   IF #AlwaysON THEN "ST10Cylinder".Cy[11].Inout.ResetOut := FALSE; END_IF;
END_REGION

REGION Network 3: CY12 interface E-NG-02NGLocationCylinder
   RUNG wire#powerrail
      Contact( #AlwaysON )
      wire#w1
      Contact( #E_stop )
      wire#w2
      Coil( "ST10Cylinder".Cy[12].In.GoWorkInterlock )
   END_RUNG
   RUNG wire#w2
      Coil( "ST10Cylinder".Cy[12].In.GoHomeInterlock )
   END_RUNG
   RUNG wire#w1
      I_Contact( #AlwaysON )
      Coil( "ST10Cylinder".Cy[12].In.Error )
   END_RUNG
   // the same network as SCL:
   "ST10Cylinder".Cy[12].In.GoWorkInterlock := #AlwaysON AND #E_stop;
   "ST10Cylinder".Cy[12].In.GoHomeInterlock := #AlwaysON AND #E_stop;
   "ST10Cylinder".Cy[12].In.Error := #AlwaysON AND NOT #AlwaysON;
END_REGION

REGION Network 4: CY13 interface F-ROOBT1Gripper1Cylinder
   RUNG wire#powerrail
      Contact( #AlwaysON )
      wire#w1
      Contact( #E_stop )
      Contact( "Robot_DB".Control.Robot1GripControl )
      wire#w2
      Coil( "ST10Cylinder".Cy[13].In.GoWorkInterlock )
   END_RUNG
   RUNG wire#w2
      Coil( "ST10Cylinder".Cy[13].In.GoHomeInterlock )
   END_RUNG
   RUNG wire#w1
      I_Contact( #AlwaysON )
      Coil( "ST10Cylinder".Cy[13].In.Error )
   END_RUNG
   // the same network as SCL:
   "ST10Cylinder".Cy[13].In.GoWorkInterlock := #AlwaysON AND #E_stop AND "Robot_DB".Control.Robot1GripControl;
   "ST10Cylinder".Cy[13].In.GoHomeInterlock := #AlwaysON AND #E_stop AND "Robot_DB".Control.Robot1GripControl;
   "ST10Cylinder".Cy[13].In.Error := #AlwaysON AND NOT #AlwaysON;
END_REGION

REGION Network 5: CY14 interface F-ROOBT1Gripper2Cylinder
   RUNG wire#powerrail
      Contact( #AlwaysON )
      wire#w1
      Contact( #E_stop )
      Contact( "Robot_DB".Control.Robot1GripControl )
      wire#w2
      Coil( "ST10Cylinder".Cy[14].In.GoWorkInterlock )
   END_RUNG
   RUNG wire#w2
      Coil( "ST10Cylinder".Cy[14].In.GoHomeInterlock )
   END_RUNG
   RUNG wire#w1
      I_Contact( #AlwaysON )
      Coil( "ST10Cylinder".Cy[14].In.Error )
   END_RUNG
   // the same network as SCL:
   "ST10Cylinder".Cy[14].In.GoWorkInterlock := #AlwaysON AND #E_stop AND "Robot_DB".Control.Robot1GripControl;
   "ST10Cylinder".Cy[14].In.GoHomeInterlock := #AlwaysON AND #E_stop AND "Robot_DB".Control.Robot1GripControl;
   "ST10Cylinder".Cy[14].In.Error := #AlwaysON AND NOT #AlwaysON;
END_REGION

REGION Network 6: CY15 interface F-ROOBT2Gripper1Cylinder
   RUNG wire#powerrail
      Contact( #AlwaysON )
      wire#w1
      Contact( #E_stop )
      Contact( "Robot_DB".Control.Robot2GripControl )
      wire#w2
      Coil( "ST10Cylinder".Cy[15].In.GoWorkInterlock )
   END_RUNG
   RUNG wire#w2
      Coil( "ST10Cylinder".Cy[15].In.GoHomeInterlock )
   END_RUNG
   RUNG wire#w1
      I_Contact( #AlwaysON )
      Coil( "ST10Cylinder".Cy[15].In.Error )
   END_RUNG
   // the same network as SCL:
   "ST10Cylinder".Cy[15].In.GoWorkInterlock := #AlwaysON AND #E_stop AND "Robot_DB".Control.Robot2GripControl;
   "ST10Cylinder".Cy[15].In.GoHomeInterlock := #AlwaysON AND #E_stop AND "Robot_DB".Control.Robot2GripControl;
   "ST10Cylinder".Cy[15].In.Error := #AlwaysON AND NOT #AlwaysON;
END_REGION

REGION Network 7: CY16 interface F-ROOBT2Gripper2Cylinder
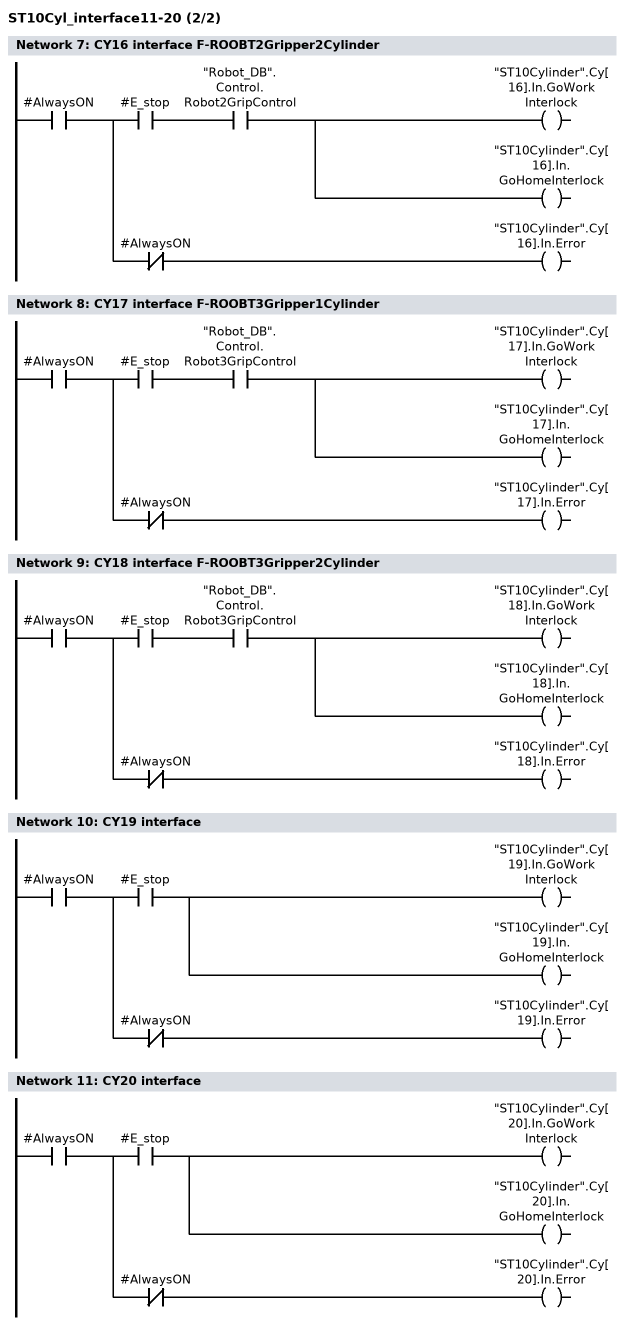
   RUNG wire#powerrail
      Contact( #AlwaysON )
      wire#w1
      Contact( #E_stop )
      Contact( "Robot_DB".Control.Robot2GripControl )
      wire#w2
      Coil( "ST10Cylinder".Cy[16].In.GoWorkInterlock )
   END_RUNG
   RUNG wire#w2
      Coil( "ST10Cylinder".Cy[16].In.GoHomeInterlock )
   END_RUNG
   RUNG wire#w1
      I_Contact( #AlwaysON )
      Coil( "ST10Cylinder".Cy[16].In.Error )
   END_RUNG
   // the same network as SCL:
   "ST10Cylinder".Cy[16].In.GoWorkInterlock := #AlwaysON AND #E_stop AND "Robot_DB".Control.Robot2GripControl;
   "ST10Cylinder".Cy[16].In.GoHomeInterlock := #AlwaysON AND #E_stop AND "Robot_DB".Control.Robot2GripControl;
   "ST10Cylinder".Cy[16].In.Error := #AlwaysON AND NOT #AlwaysON;
END_REGION

REGION Network 8: CY17 interface F-ROOBT3Gripper1Cylinder
   RUNG wire#powerrail
      Contact( #AlwaysON )
      wire#w1
      Contact( #E_stop )
      Contact( "Robot_DB".Control.Robot3GripControl )
      wire#w2
      Coil( "ST10Cylinder".Cy[17].In.GoWorkInterlock )
   END_RUNG
   RUNG wire#w2
      Coil( "ST10Cylinder".Cy[17].In.GoHomeInterlock )
   END_RUNG
   RUNG wire#w1
      I_Contact( #AlwaysON )
      Coil( "ST10Cylinder".Cy[17].In.Error )
   END_RUNG
   // the same network as SCL:
   "ST10Cylinder".Cy[17].In.GoWorkInterlock := #AlwaysON AND #E_stop AND "Robot_DB".Control.Robot3GripControl;
   "ST10Cylinder".Cy[17].In.GoHomeInterlock := #AlwaysON AND #E_stop AND "Robot_DB".Control.Robot3GripControl;
   "ST10Cylinder".Cy[17].In.Error := #AlwaysON AND NOT #AlwaysON;
END_REGION

REGION Network 9: CY18 interface F-ROOBT3Gripper2Cylinder
   RUNG wire#powerrail
      Contact( #AlwaysON )
      wire#w1
      Contact( #E_stop )
      Contact( "Robot_DB".Control.Robot3GripControl )
      wire#w2
      Coil( "ST10Cylinder".Cy[18].In.GoWorkInterlock )
   END_RUNG
   RUNG wire#w2
      Coil( "ST10Cylinder".Cy[18].In.GoHomeInterlock )
   END_RUNG
   RUNG wire#w1
      I_Contact( #AlwaysON )
      Coil( "ST10Cylinder".Cy[18].In.Error )
   END_RUNG
   // the same network as SCL:
   "ST10Cylinder".Cy[18].In.GoWorkInterlock := #AlwaysON AND #E_stop AND "Robot_DB".Control.Robot3GripControl;
   "ST10Cylinder".Cy[18].In.GoHomeInterlock := #AlwaysON AND #E_stop AND "Robot_DB".Control.Robot3GripControl;
   "ST10Cylinder".Cy[18].In.Error := #AlwaysON AND NOT #AlwaysON;
END_REGION

REGION Network 10: CY19 interface
   RUNG wire#powerrail
      Contact( #AlwaysON )
      wire#w1
      Contact( #E_stop )
      wire#w2
      Coil( "ST10Cylinder".Cy[19].In.GoWorkInterlock )
   END_RUNG
   RUNG wire#w2
      Coil( "ST10Cylinder".Cy[19].In.GoHomeInterlock )
   END_RUNG
   RUNG wire#w1
      I_Contact( #AlwaysON )
      Coil( "ST10Cylinder".Cy[19].In.Error )
   END_RUNG
   // the same network as SCL:
   "ST10Cylinder".Cy[19].In.GoWorkInterlock := #AlwaysON AND #E_stop;
   "ST10Cylinder".Cy[19].In.GoHomeInterlock := #AlwaysON AND #E_stop;
   "ST10Cylinder".Cy[19].In.Error := #AlwaysON AND NOT #AlwaysON;
END_REGION

REGION Network 11: CY20 interface
   RUNG wire#powerrail
      Contact( #AlwaysON )
      wire#w1
      Contact( #E_stop )
      wire#w2
      Coil( "ST10Cylinder".Cy[20].In.GoWorkInterlock )
   END_RUNG
   RUNG wire#w2
      Coil( "ST10Cylinder".Cy[20].In.GoHomeInterlock )
   END_RUNG
   RUNG wire#w1
      I_Contact( #AlwaysON )
      Coil( "ST10Cylinder".Cy[20].In.Error )
   END_RUNG
   // the same network as SCL:
   "ST10Cylinder".Cy[20].In.GoWorkInterlock := #AlwaysON AND #E_stop;
   "ST10Cylinder".Cy[20].In.GoHomeInterlock := #AlwaysON AND #E_stop;
   "ST10Cylinder".Cy[20].In.Error := #AlwaysON AND NOT #AlwaysON;
END_REGION
END_FUNCTION

FUNCTION "ST10Cyl_interface21-30" : Void   // FC1022, LAD
{ S7_Optimized_Access := 'FALSE' }
// stored: AutoNumber false, SetENOAutomatically false
   VAR_INPUT
      AlwaysON : Bool;
      E_stop : Bool;
   END_VAR
   VAR_TEMP
      tTest : Bool;
   END_VAR
BEGIN

REGION Network 1 (SCL): Cylinder 21-30 IO Interface (SCL)

   //Cylinder21 IO  H-shaftLiftingLiftingCylinder
   //Input
   "ST10Cylinder".Cy[21].In.WorkPositionSensor := "iH-shaftLiftingLiftingCylinderInWP" ;
   "ST10Cylinder".Cy[21].In.HomePositionSensor := "iH-shaftLiftingLiftingCylinderInHP" ;
   //Output
   "oH-shaftLiftingLiftingCylinderToWP" := "ST10Cylinder".Cy[21].Out.GoWorkPosition;
   "oH-shaftLiftingLiftingCylinderToHP" := "ST10Cylinder".Cy[21].Out.GoHomePosition;

   //Cylinder22 IO  H-shaftLiftingPalletLocationCylinder
   //Input
   "ST10Cylinder".Cy[22].In.WorkPositionSensor := "iH-shaftLiftingPalletLocationCylinderInWP" ;
   "ST10Cylinder".Cy[22].In.HomePositionSensor :="iH-shaftLiftingPalletLocationCylinderInHP"  ;
   //Output
   "oH-shaftLiftingPalletLocationCylinderToWP" := "ST10Cylinder".Cy[22].Out.GoWorkPosition;
   "oH-shaftLiftingPalletLocationCylinderToHP" := "ST10Cylinder".Cy[22].Out.GoHomePosition;

   //Cylinder23 IO  H-shaftLoadingStopperCylinder1
   //Input
   "ST10Cylinder".Cy[23].In.WorkPositionSensor := "oH-shaftLoadingStopperCylinder1_ToWP";
   "ST10Cylinder".Cy[23].In.HomePositionSensor := "oH-shaftLoadingStopperCylinder1_ToHP" ;
   //Output
   "oH-shaftLoadingStopperCylinder1_ToWP" := "ST10Cylinder".Cy[23].Out.GoWorkPosition;
   "oH-shaftLoadingStopperCylinder1_ToHP" := "ST10Cylinder".Cy[23].Out.GoHomePosition;

   //Cylinder24 IO  H-shaftLoadingStopperCylinder2
   //Input
   "ST10Cylinder".Cy[24].In.WorkPositionSensor := "oH-shaftLoadingStopperCylinder2_ToWP" ;
   "ST10Cylinder".Cy[24].In.HomePositionSensor := "oH-shaftLoadingStopperCylinder2_ToHP";
   //Output
   "oH-shaftLoadingStopperCylinder2_ToWP" := "ST10Cylinder".Cy[24].Out.GoWorkPosition;
   "oH-shaftLoadingStopperCylinder2_ToHP" := "ST10Cylinder".Cy[24].Out.GoHomePosition;

   //Cylinder25 IO  H-shaftLoadingStopperCylinder3
   //Input
   "ST10Cylinder".Cy[25].In.WorkPositionSensor := "oH-shaftLoadingStopperCylinder3_ToWP";
   "ST10Cylinder".Cy[25].In.HomePositionSensor := "oH-shaftLoadingStopperCylinder3_ToHP";
   //Output
   "oH-shaftLoadingStopperCylinder3_ToWP" := "ST10Cylinder".Cy[25].Out.GoWorkPosition;
   "oH-shaftLoadingStopperCylinder3_ToHP" := "ST10Cylinder".Cy[25].Out.GoHomePosition;

   //Cylinder26 H-shaftLoadingStopperCylinder4
   //Input
   "ST10Cylinder".Cy[26].In.WorkPositionSensor := "oH-shaftLoadingStopperCylinder4_ToWP";
   "ST10Cylinder".Cy[26].In.HomePositionSensor := "oH-shaftLoadingStopperCylinder4_ToHP" ;
   //Output
   "oH-shaftLoadingStopperCylinder4_ToWP" := "ST10Cylinder".Cy[26].Out.GoWorkPosition;
   "oH-shaftLoadingStopperCylinder4_ToHP" := "ST10Cylinder".Cy[26].Out.GoHomePosition;

   //Cylinder27 H-shaftTakeStopperCylinder1
   //Input
   "ST10Cylinder".Cy[27].In.WorkPositionSensor :="oH-shaftTakeStopperCylinder1_ToWP" ;
   "ST10Cylinder".Cy[27].In.HomePositionSensor :="oH-shaftTakeStopperCylinder1_ToHP";
   //Output
   "oH-shaftTakeStopperCylinder1_ToWP" :="ST10Cylinder".Cy[27].Out.GoWorkPosition;
   "oH-shaftTakeStopperCylinder1_ToHP" := "ST10Cylinder".Cy[27].Out.GoHomePosition;

   //Cylinder28 H-shaftTakeStopperCylinder2
   //Input
   "ST10Cylinder".Cy[28].In.WorkPositionSensor :="oH-shaftTakeStopperCylinder2_ToWP" ;
   "ST10Cylinder".Cy[28].In.HomePositionSensor := "oH-shaftTakeStopperCylinder2_ToHP";
   //Output
   "oH-shaftTakeStopperCylinder2_ToWP" := "ST10Cylinder".Cy[28].Out.GoWorkPosition;
   "oH-shaftTakeStopperCylinder2_ToHP" := "ST10Cylinder".Cy[28].Out.GoHomePosition;

   //Cylinder29 H-shaftTakeStopperCylinder3
   //Input
   "ST10Cylinder".Cy[29].In.WorkPositionSensor :="oH-shaftTakeStopperCylinder3_ToWP" ;
   "ST10Cylinder".Cy[29].In.HomePositionSensor :="oH-shaftTakeStopperCylinder3_ToHP";
   //Output
   "oH-shaftTakeStopperCylinder3_ToWP" := "ST10Cylinder".Cy[29].Out.GoWorkPosition;
   "oH-shaftTakeStopperCylinder3_ToHP" := "ST10Cylinder".Cy[29].Out.GoHomePosition;

    (*
    //Cylinder30 H-shaftLoadingStopperCylinder4_2  
   // //Input
   "ST10Cylinder".Cy[30].In.WorkPositionSensor := "oH-shaftLoadingStopperCylinder4_2";
   "ST10Cylinder".Cy[30].In.HomePositionSensor := NOT "oH-shaftLoadingStopperCylinder4_2";
   // //Output
    "oH-shaftLoadingStopperCylinder4_2" := "ST10Cylinder".Cy[30].Out.GoWorkPosition;
    "Feeding washer  lift Cylinder ToHP" := "ST10Cylinder".Cy[30].Out.GoHomePosition;
   *)
END_REGION

REGION Network 2: CY21 interface H-shaftLiftingLiftingCylinder
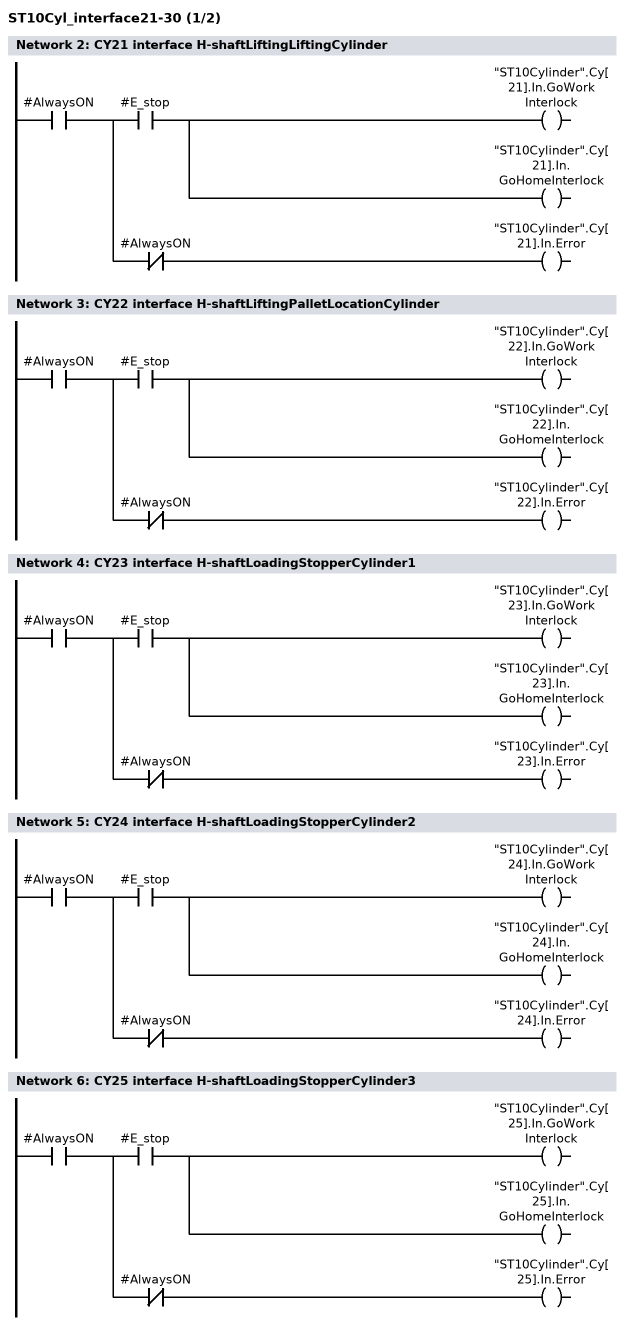
   RUNG wire#powerrail
      Contact( #AlwaysON )
      wire#w1
      Contact( #E_stop )
      wire#w2
      Coil( "ST10Cylinder".Cy[21].In.GoWorkInterlock )
   END_RUNG
   RUNG wire#w2
      Coil( "ST10Cylinder".Cy[21].In.GoHomeInterlock )
   END_RUNG
   RUNG wire#w1
      I_Contact( #AlwaysON )
      Coil( "ST10Cylinder".Cy[21].In.Error )
   END_RUNG
   // the same network as SCL:
   "ST10Cylinder".Cy[21].In.GoWorkInterlock := #AlwaysON AND #E_stop;
   "ST10Cylinder".Cy[21].In.GoHomeInterlock := #AlwaysON AND #E_stop;
   "ST10Cylinder".Cy[21].In.Error := #AlwaysON AND NOT #AlwaysON;
END_REGION

REGION Network 3: CY22 interface H-shaftLiftingPalletLocationCylinder
   RUNG wire#powerrail
      Contact( #AlwaysON )
      wire#w1
      Contact( #E_stop )
      wire#w2
      Coil( "ST10Cylinder".Cy[22].In.GoWorkInterlock )
   END_RUNG
   RUNG wire#w2
      Coil( "ST10Cylinder".Cy[22].In.GoHomeInterlock )
   END_RUNG
   RUNG wire#w1
      I_Contact( #AlwaysON )
      Coil( "ST10Cylinder".Cy[22].In.Error )
   END_RUNG
   // the same network as SCL:
   "ST10Cylinder".Cy[22].In.GoWorkInterlock := #AlwaysON AND #E_stop;
   "ST10Cylinder".Cy[22].In.GoHomeInterlock := #AlwaysON AND #E_stop;
   "ST10Cylinder".Cy[22].In.Error := #AlwaysON AND NOT #AlwaysON;
END_REGION

REGION Network 4: CY23 interface H-shaftLoadingStopperCylinder1
   RUNG wire#powerrail
      Contact( #AlwaysON )
      wire#w1
      Contact( #E_stop )
      wire#w2
      Coil( "ST10Cylinder".Cy[23].In.GoWorkInterlock )
   END_RUNG
   RUNG wire#w2
      Coil( "ST10Cylinder".Cy[23].In.GoHomeInterlock )
   END_RUNG
   RUNG wire#w1
      I_Contact( #AlwaysON )
      Coil( "ST10Cylinder".Cy[23].In.Error )
   END_RUNG
   // the same network as SCL:
   "ST10Cylinder".Cy[23].In.GoWorkInterlock := #AlwaysON AND #E_stop;
   "ST10Cylinder".Cy[23].In.GoHomeInterlock := #AlwaysON AND #E_stop;
   "ST10Cylinder".Cy[23].In.Error := #AlwaysON AND NOT #AlwaysON;
END_REGION

REGION Network 5: CY24 interface H-shaftLoadingStopperCylinder2
   RUNG wire#powerrail
      Contact( #AlwaysON )
      wire#w1
      Contact( #E_stop )
      wire#w2
      Coil( "ST10Cylinder".Cy[24].In.GoWorkInterlock )
   END_RUNG
   RUNG wire#w2
      Coil( "ST10Cylinder".Cy[24].In.GoHomeInterlock )
   END_RUNG
   RUNG wire#w1
      I_Contact( #AlwaysON )
      Coil( "ST10Cylinder".Cy[24].In.Error )
   END_RUNG
   // the same network as SCL:
   "ST10Cylinder".Cy[24].In.GoWorkInterlock := #AlwaysON AND #E_stop;
   "ST10Cylinder".Cy[24].In.GoHomeInterlock := #AlwaysON AND #E_stop;
   "ST10Cylinder".Cy[24].In.Error := #AlwaysON AND NOT #AlwaysON;
END_REGION

REGION Network 6: CY25 interface H-shaftLoadingStopperCylinder3
   RUNG wire#powerrail
      Contact( #AlwaysON )
      wire#w1
      Contact( #E_stop )
      wire#w2
      Coil( "ST10Cylinder".Cy[25].In.GoWorkInterlock )
   END_RUNG
   RUNG wire#w2
      Coil( "ST10Cylinder".Cy[25].In.GoHomeInterlock )
   END_RUNG
   RUNG wire#w1
      I_Contact( #AlwaysON )
      Coil( "ST10Cylinder".Cy[25].In.Error )
   END_RUNG
   // the same network as SCL:
   "ST10Cylinder".Cy[25].In.GoWorkInterlock := #AlwaysON AND #E_stop;
   "ST10Cylinder".Cy[25].In.GoHomeInterlock := #AlwaysON AND #E_stop;
   "ST10Cylinder".Cy[25].In.Error := #AlwaysON AND NOT #AlwaysON;
END_REGION

REGION Network 7: CY26 interface H-shaftLoadingStopperCylinder4
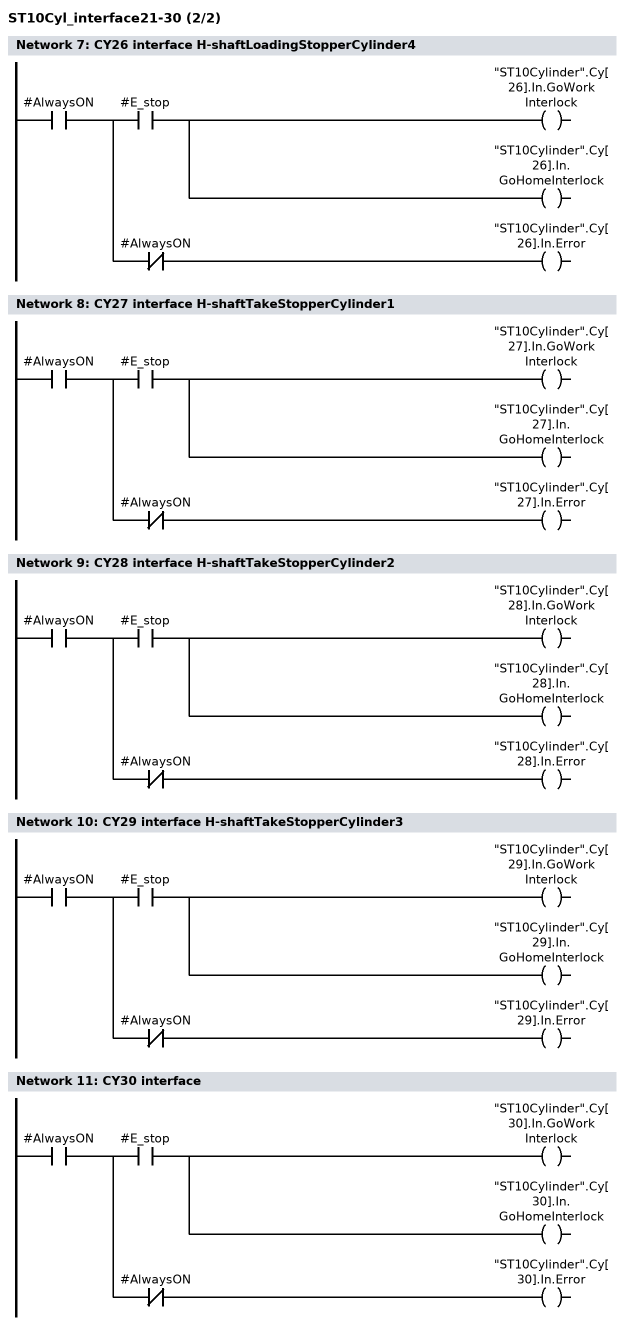
   RUNG wire#powerrail
      Contact( #AlwaysON )
      wire#w1
      Contact( #E_stop )
      wire#w2
      Coil( "ST10Cylinder".Cy[26].In.GoWorkInterlock )
   END_RUNG
   RUNG wire#w2
      Coil( "ST10Cylinder".Cy[26].In.GoHomeInterlock )
   END_RUNG
   RUNG wire#w1
      I_Contact( #AlwaysON )
      Coil( "ST10Cylinder".Cy[26].In.Error )
   END_RUNG
   // the same network as SCL:
   "ST10Cylinder".Cy[26].In.GoWorkInterlock := #AlwaysON AND #E_stop;
   "ST10Cylinder".Cy[26].In.GoHomeInterlock := #AlwaysON AND #E_stop;
   "ST10Cylinder".Cy[26].In.Error := #AlwaysON AND NOT #AlwaysON;
END_REGION

REGION Network 8: CY27 interface H-shaftTakeStopperCylinder1
   RUNG wire#powerrail
      Contact( #AlwaysON )
      wire#w1
      Contact( #E_stop )
      wire#w2
      Coil( "ST10Cylinder".Cy[27].In.GoWorkInterlock )
   END_RUNG
   RUNG wire#w2
      Coil( "ST10Cylinder".Cy[27].In.GoHomeInterlock )
   END_RUNG
   RUNG wire#w1
      I_Contact( #AlwaysON )
      Coil( "ST10Cylinder".Cy[27].In.Error )
   END_RUNG
   // the same network as SCL:
   "ST10Cylinder".Cy[27].In.GoWorkInterlock := #AlwaysON AND #E_stop;
   "ST10Cylinder".Cy[27].In.GoHomeInterlock := #AlwaysON AND #E_stop;
   "ST10Cylinder".Cy[27].In.Error := #AlwaysON AND NOT #AlwaysON;
END_REGION

REGION Network 9: CY28 interface H-shaftTakeStopperCylinder2
   RUNG wire#powerrail
      Contact( #AlwaysON )
      wire#w1
      Contact( #E_stop )
      wire#w2
      Coil( "ST10Cylinder".Cy[28].In.GoWorkInterlock )
   END_RUNG
   RUNG wire#w2
      Coil( "ST10Cylinder".Cy[28].In.GoHomeInterlock )
   END_RUNG
   RUNG wire#w1
      I_Contact( #AlwaysON )
      Coil( "ST10Cylinder".Cy[28].In.Error )
   END_RUNG
   // the same network as SCL:
   "ST10Cylinder".Cy[28].In.GoWorkInterlock := #AlwaysON AND #E_stop;
   "ST10Cylinder".Cy[28].In.GoHomeInterlock := #AlwaysON AND #E_stop;
   "ST10Cylinder".Cy[28].In.Error := #AlwaysON AND NOT #AlwaysON;
END_REGION

REGION Network 10: CY29 interface H-shaftTakeStopperCylinder3
   RUNG wire#powerrail
      Contact( #AlwaysON )
      wire#w1
      Contact( #E_stop )
      wire#w2
      Coil( "ST10Cylinder".Cy[29].In.GoWorkInterlock )
   END_RUNG
   RUNG wire#w2
      Coil( "ST10Cylinder".Cy[29].In.GoHomeInterlock )
   END_RUNG
   RUNG wire#w1
      I_Contact( #AlwaysON )
      Coil( "ST10Cylinder".Cy[29].In.Error )
   END_RUNG
   // the same network as SCL:
   "ST10Cylinder".Cy[29].In.GoWorkInterlock := #AlwaysON AND #E_stop;
   "ST10Cylinder".Cy[29].In.GoHomeInterlock := #AlwaysON AND #E_stop;
   "ST10Cylinder".Cy[29].In.Error := #AlwaysON AND NOT #AlwaysON;
END_REGION

REGION Network 11: CY30 interface
   RUNG wire#powerrail
      Contact( #AlwaysON )
      wire#w1
      Contact( #E_stop )
      wire#w2
      Coil( "ST10Cylinder".Cy[30].In.GoWorkInterlock )
   END_RUNG
   RUNG wire#w2
      Coil( "ST10Cylinder".Cy[30].In.GoHomeInterlock )
   END_RUNG
   RUNG wire#w1
      I_Contact( #AlwaysON )
      Coil( "ST10Cylinder".Cy[30].In.Error )
   END_RUNG
   // the same network as SCL:
   "ST10Cylinder".Cy[30].In.GoWorkInterlock := #AlwaysON AND #E_stop;
   "ST10Cylinder".Cy[30].In.GoHomeInterlock := #AlwaysON AND #E_stop;
   "ST10Cylinder".Cy[30].In.Error := #AlwaysON AND NOT #AlwaysON;
END_REGION
END_FUNCTION

FUNCTION "ST10Cyl_interface31-40" : Void   // FC1023, LAD
{ S7_Optimized_Access := 'FALSE' }
// stored: AutoNumber false, SetENOAutomatically false
   VAR_INPUT
      AlwaysON : Bool;
      E_stop : Bool;
   END_VAR
   VAR_TEMP
      tTest : Bool;
   END_VAR
BEGIN

REGION Network 1 (SCL): Cylinder 31-40 IO Interface (SCL)

   //Cylinder31 IO  J-magnetLiftingLiftingCylinder
   //Input
   "ST10Cylinder".Cy[31].In.WorkPositionSensor := "iJ-magnetLiftingLiftingCylinderInWP";
   "ST10Cylinder".Cy[31].In.HomePositionSensor := "iJ-magnetLiftingLiftingCylinderInHP";
   //Output
   "oJ-magnetLiftingLiftingCylinderToWP" := "ST10Cylinder".Cy[31].Out.GoWorkPosition;
   "oJ-magnetLiftingLiftingCylinderToHP" := "ST10Cylinder".Cy[31].Out.GoHomePosition;

   //Cylinder32 IO  J-magnetLiftingPalletLocationCylinder
   //Input
   "ST10Cylinder".Cy[32].In.WorkPositionSensor := "iJ-magnetLiftingPalletLocationCylinderInWP";
   "ST10Cylinder".Cy[32].In.HomePositionSensor := "iJ-magnetLiftingPalletLocationCylinderInHP";
   //Output
   "oJ-magnetLiftingPalletLocationCylinderToWP" := "ST10Cylinder".Cy[32].Out.GoWorkPosition;
   "oJ-magnetLiftingPalletLocationCylinderToHP" := "ST10Cylinder".Cy[32].Out.GoHomePosition;

   //Cylinder33 IO  J-magnetLoadingStopperCylinder1
   //Input
   "ST10Cylinder".Cy[33].In.WorkPositionSensor := "oJ-magnetLoadingStopperCylinder1_ToWP";
   "ST10Cylinder".Cy[33].In.HomePositionSensor := "oJ-magnetLoadingStopperCylinder1_ToHP";
   //Output
   "oJ-magnetLoadingStopperCylinder1_ToWP" := "ST10Cylinder".Cy[33].Out.GoWorkPosition;
   "oJ-magnetLoadingStopperCylinder1_ToHP" := "ST10Cylinder".Cy[33].Out.GoHomePosition;

   //Cylinder34 IO  J-magnetLoadingStopperCylinder2
   //Input
   "ST10Cylinder".Cy[34].In.WorkPositionSensor := "oJ-magnetLoadingStopperCylinder2_ToWP";
   "ST10Cylinder".Cy[34].In.HomePositionSensor := "oJ-magnetLoadingStopperCylinder2_ToHP";
   //Output
   "oJ-magnetLoadingStopperCylinder2_ToWP" := "ST10Cylinder".Cy[34].Out.GoWorkPosition;
   "oJ-magnetLoadingStopperCylinder2_ToHP" := "ST10Cylinder".Cy[34].Out.GoHomePosition;

   //Cylinder35 IO  J-magnetLoadingStopperCylinder3
   //Input
   "ST10Cylinder".Cy[35].In.WorkPositionSensor := "oJ-magnetLoadingStopperCylinder3_ToWP";
   "ST10Cylinder".Cy[35].In.HomePositionSensor := "oJ-magnetLoadingStopperCylinder3_ToHP";
   //Output
   "oJ-magnetLoadingStopperCylinder3_ToWP" := "ST10Cylinder".Cy[35].Out.GoWorkPosition;
   "oJ-magnetLoadingStopperCylinder3_ToHP" := "ST10Cylinder".Cy[35].Out.GoHomePosition;

   //Cylinder36 J-magnetLoadingStopperCylinder4
   //Input
   "ST10Cylinder".Cy[36].In.WorkPositionSensor := "oJ-magnetLoadingStopperCylinder4_ToWP";
   "ST10Cylinder".Cy[36].In.HomePositionSensor := "oJ-magnetLoadingStopperCylinder4_ToHP";
   //Output
   "oJ-magnetLoadingStopperCylinder4_ToWP" := "ST10Cylinder".Cy[36].Out.GoWorkPosition;
   "oJ-magnetLoadingStopperCylinder4_ToHP" := "ST10Cylinder".Cy[36].Out.GoHomePosition;

   //Cylinder37 J-magnetTakeStopperCylinder1
   //Input
   "ST10Cylinder".Cy[37].In.WorkPositionSensor := "oJ-magnetTakeStopperCylinder1_ToWP";
   "ST10Cylinder".Cy[37].In.HomePositionSensor := "oJ-magnetTakeStopperCylinder1_ToHP";
   //Output
   "oJ-magnetTakeStopperCylinder1_ToWP" := "ST10Cylinder".Cy[37].Out.GoWorkPosition;
   "oJ-magnetTakeStopperCylinder1_ToHP" := "ST10Cylinder".Cy[37].Out.GoHomePosition;

   //Cylinder38 J-magnetTakeStopperCylinder2
   //Input
   "ST10Cylinder".Cy[38].In.WorkPositionSensor := "oJ-magnetTakeStopperCylinder2_ToWP";
   "ST10Cylinder".Cy[38].In.HomePositionSensor := "oJ-magnetTakeStopperCylinder2_ToHP";
   //Output
   "oJ-magnetTakeStopperCylinder2_ToWP" := "ST10Cylinder".Cy[38].Out.GoWorkPosition;
   "oJ-magnetTakeStopperCylinder2_ToHP" := "ST10Cylinder".Cy[38].Out.GoHomePosition;

   //Cylinder39 J-magnetTakeStopperCylinder3
   //Input
   "ST10Cylinder".Cy[39].In.WorkPositionSensor := "oJ-magnetTakeStopperCylinder3_ToWP";
   "ST10Cylinder".Cy[39].In.HomePositionSensor := "oJ-magnetTakeStopperCylinder3_ToHP";
   //Output
   "oJ-magnetTakeStopperCylinder3_ToWP" := "ST10Cylinder".Cy[39].Out.GoWorkPosition;
   "oJ-magnetTakeStopperCylinder3_ToHP" := "ST10Cylinder".Cy[39].Out.GoHomePosition;

   (*
   //Cylinder40 J-magnetLoadingStopperCylinder4_2
   // //Input
   "ST10Cylinder".Cy[40].In.WorkPositionSensor := "oJ-magnetLoadingStopperCylinder4_2";
   "ST10Cylinder".Cy[40].In.HomePositionSensor := NOT "oJ-magnetLoadingStopperCylinder4_2";
   // //Output
   "oJ-magnetLoadingStopperCylinder4_2" := "ST10Cylinder".Cy[40].Out.GoWorkPosition;
   "Feeding washer  lift Cylinder ToHP" := "ST10Cylinder".Cy[40].Out.GoHomePosition;
   *)
END_REGION

REGION Network 2: CY31 interface J-magnetLiftingLiftingCylinder
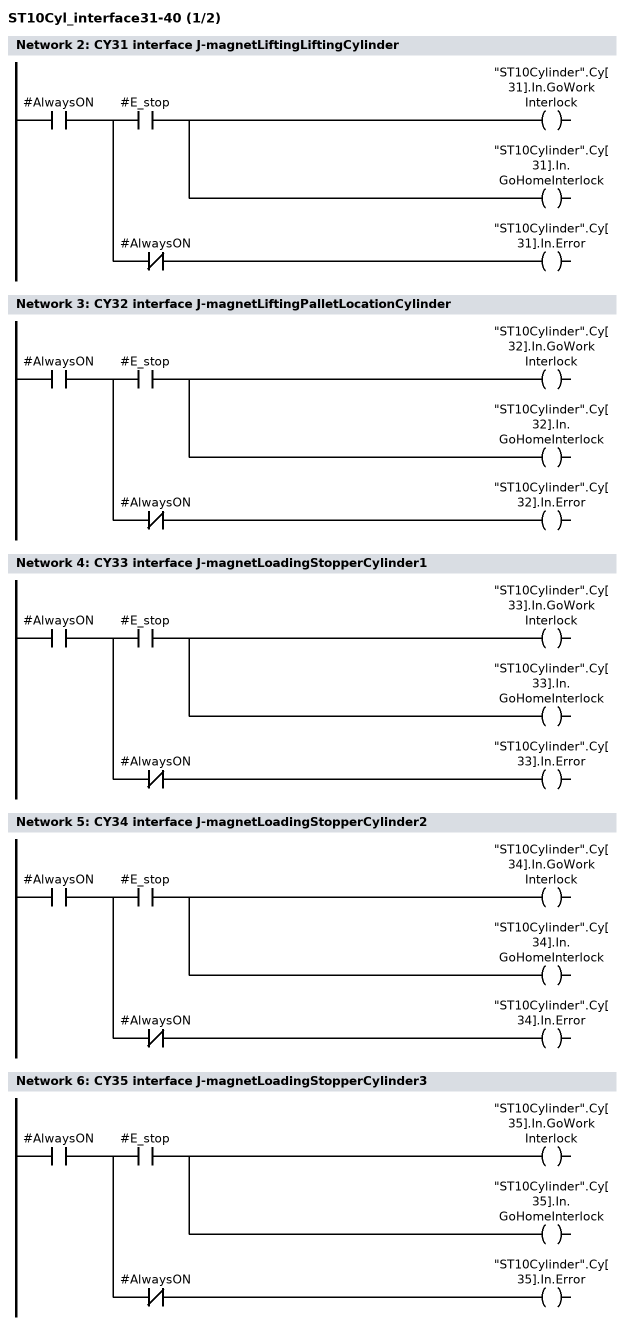
   RUNG wire#powerrail
      Contact( #AlwaysON )
      wire#w1
      Contact( #E_stop )
      wire#w2
      Coil( "ST10Cylinder".Cy[31].In.GoWorkInterlock )
   END_RUNG
   RUNG wire#w2
      Coil( "ST10Cylinder".Cy[31].In.GoHomeInterlock )
   END_RUNG
   RUNG wire#w1
      I_Contact( #AlwaysON )
      Coil( "ST10Cylinder".Cy[31].In.Error )
   END_RUNG
   // the same network as SCL:
   "ST10Cylinder".Cy[31].In.GoWorkInterlock := #AlwaysON AND #E_stop;
   "ST10Cylinder".Cy[31].In.GoHomeInterlock := #AlwaysON AND #E_stop;
   "ST10Cylinder".Cy[31].In.Error := #AlwaysON AND NOT #AlwaysON;
END_REGION

REGION Network 3: CY32 interface J-magnetLiftingPalletLocationCylinder
   RUNG wire#powerrail
      Contact( #AlwaysON )
      wire#w1
      Contact( #E_stop )
      wire#w2
      Coil( "ST10Cylinder".Cy[32].In.GoWorkInterlock )
   END_RUNG
   RUNG wire#w2
      Coil( "ST10Cylinder".Cy[32].In.GoHomeInterlock )
   END_RUNG
   RUNG wire#w1
      I_Contact( #AlwaysON )
      Coil( "ST10Cylinder".Cy[32].In.Error )
   END_RUNG
   // the same network as SCL:
   "ST10Cylinder".Cy[32].In.GoWorkInterlock := #AlwaysON AND #E_stop;
   "ST10Cylinder".Cy[32].In.GoHomeInterlock := #AlwaysON AND #E_stop;
   "ST10Cylinder".Cy[32].In.Error := #AlwaysON AND NOT #AlwaysON;
END_REGION

REGION Network 4: CY33 interface J-magnetLoadingStopperCylinder1
   RUNG wire#powerrail
      Contact( #AlwaysON )
      wire#w1
      Contact( #E_stop )
      wire#w2
      Coil( "ST10Cylinder".Cy[33].In.GoWorkInterlock )
   END_RUNG
   RUNG wire#w2
      Coil( "ST10Cylinder".Cy[33].In.GoHomeInterlock )
   END_RUNG
   RUNG wire#w1
      I_Contact( #AlwaysON )
      Coil( "ST10Cylinder".Cy[33].In.Error )
   END_RUNG
   // the same network as SCL:
   "ST10Cylinder".Cy[33].In.GoWorkInterlock := #AlwaysON AND #E_stop;
   "ST10Cylinder".Cy[33].In.GoHomeInterlock := #AlwaysON AND #E_stop;
   "ST10Cylinder".Cy[33].In.Error := #AlwaysON AND NOT #AlwaysON;
END_REGION

REGION Network 5: CY34 interface J-magnetLoadingStopperCylinder2
   RUNG wire#powerrail
      Contact( #AlwaysON )
      wire#w1
      Contact( #E_stop )
      wire#w2
      Coil( "ST10Cylinder".Cy[34].In.GoWorkInterlock )
   END_RUNG
   RUNG wire#w2
      Coil( "ST10Cylinder".Cy[34].In.GoHomeInterlock )
   END_RUNG
   RUNG wire#w1
      I_Contact( #AlwaysON )
      Coil( "ST10Cylinder".Cy[34].In.Error )
   END_RUNG
   // the same network as SCL:
   "ST10Cylinder".Cy[34].In.GoWorkInterlock := #AlwaysON AND #E_stop;
   "ST10Cylinder".Cy[34].In.GoHomeInterlock := #AlwaysON AND #E_stop;
   "ST10Cylinder".Cy[34].In.Error := #AlwaysON AND NOT #AlwaysON;
END_REGION

REGION Network 6: CY35 interface J-magnetLoadingStopperCylinder3
   RUNG wire#powerrail
      Contact( #AlwaysON )
      wire#w1
      Contact( #E_stop )
      wire#w2
      Coil( "ST10Cylinder".Cy[35].In.GoWorkInterlock )
   END_RUNG
   RUNG wire#w2
      Coil( "ST10Cylinder".Cy[35].In.GoHomeInterlock )
   END_RUNG
   RUNG wire#w1
      I_Contact( #AlwaysON )
      Coil( "ST10Cylinder".Cy[35].In.Error )
   END_RUNG
   // the same network as SCL:
   "ST10Cylinder".Cy[35].In.GoWorkInterlock := #AlwaysON AND #E_stop;
   "ST10Cylinder".Cy[35].In.GoHomeInterlock := #AlwaysON AND #E_stop;
   "ST10Cylinder".Cy[35].In.Error := #AlwaysON AND NOT #AlwaysON;
END_REGION

REGION Network 7: CY36 interface J-magnetLoadingStopperCylinder4
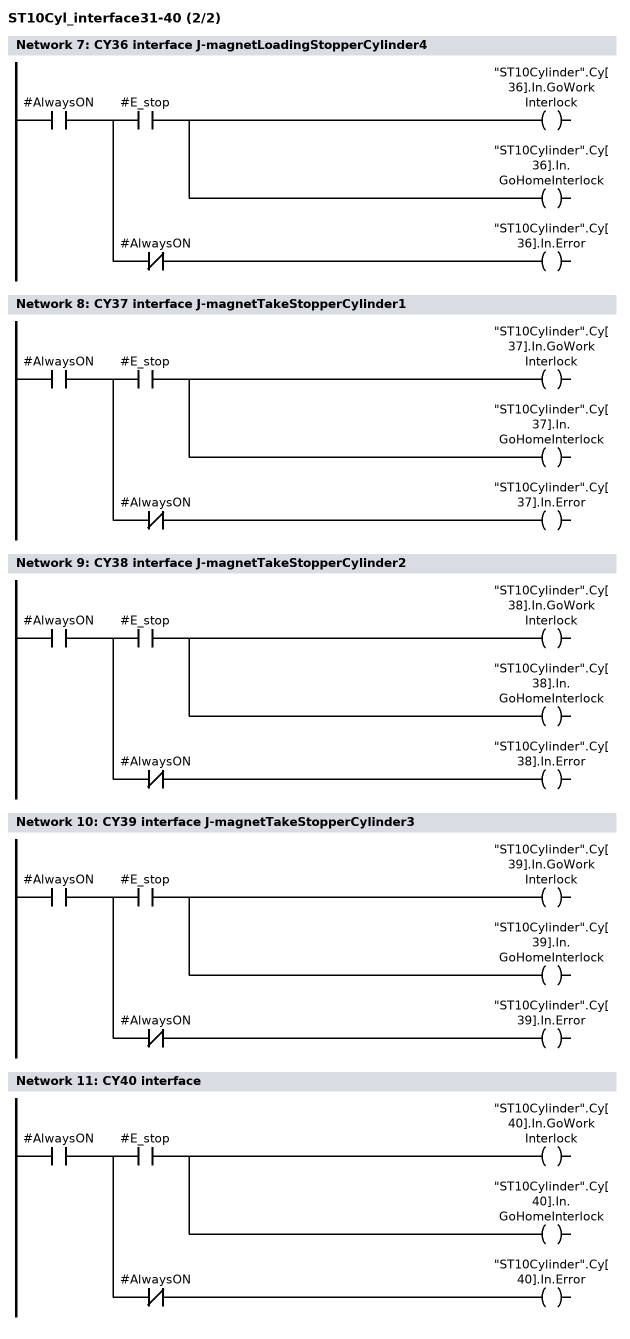
   RUNG wire#powerrail
      Contact( #AlwaysON )
      wire#w1
      Contact( #E_stop )
      wire#w2
      Coil( "ST10Cylinder".Cy[36].In.GoWorkInterlock )
   END_RUNG
   RUNG wire#w2
      Coil( "ST10Cylinder".Cy[36].In.GoHomeInterlock )
   END_RUNG
   RUNG wire#w1
      I_Contact( #AlwaysON )
      Coil( "ST10Cylinder".Cy[36].In.Error )
   END_RUNG
   // the same network as SCL:
   "ST10Cylinder".Cy[36].In.GoWorkInterlock := #AlwaysON AND #E_stop;
   "ST10Cylinder".Cy[36].In.GoHomeInterlock := #AlwaysON AND #E_stop;
   "ST10Cylinder".Cy[36].In.Error := #AlwaysON AND NOT #AlwaysON;
END_REGION

REGION Network 8: CY37 interface J-magnetTakeStopperCylinder1
   RUNG wire#powerrail
      Contact( #AlwaysON )
      wire#w1
      Contact( #E_stop )
      wire#w2
      Coil( "ST10Cylinder".Cy[37].In.GoWorkInterlock )
   END_RUNG
   RUNG wire#w2
      Coil( "ST10Cylinder".Cy[37].In.GoHomeInterlock )
   END_RUNG
   RUNG wire#w1
      I_Contact( #AlwaysON )
      Coil( "ST10Cylinder".Cy[37].In.Error )
   END_RUNG
   // the same network as SCL:
   "ST10Cylinder".Cy[37].In.GoWorkInterlock := #AlwaysON AND #E_stop;
   "ST10Cylinder".Cy[37].In.GoHomeInterlock := #AlwaysON AND #E_stop;
   "ST10Cylinder".Cy[37].In.Error := #AlwaysON AND NOT #AlwaysON;
END_REGION

REGION Network 9: CY38 interface J-magnetTakeStopperCylinder2
   RUNG wire#powerrail
      Contact( #AlwaysON )
      wire#w1
      Contact( #E_stop )
      wire#w2
      Coil( "ST10Cylinder".Cy[38].In.GoWorkInterlock )
   END_RUNG
   RUNG wire#w2
      Coil( "ST10Cylinder".Cy[38].In.GoHomeInterlock )
   END_RUNG
   RUNG wire#w1
      I_Contact( #AlwaysON )
      Coil( "ST10Cylinder".Cy[38].In.Error )
   END_RUNG
   // the same network as SCL:
   "ST10Cylinder".Cy[38].In.GoWorkInterlock := #AlwaysON AND #E_stop;
   "ST10Cylinder".Cy[38].In.GoHomeInterlock := #AlwaysON AND #E_stop;
   "ST10Cylinder".Cy[38].In.Error := #AlwaysON AND NOT #AlwaysON;
END_REGION

REGION Network 10: CY39 interface J-magnetTakeStopperCylinder3
   RUNG wire#powerrail
      Contact( #AlwaysON )
      wire#w1
      Contact( #E_stop )
      wire#w2
      Coil( "ST10Cylinder".Cy[39].In.GoWorkInterlock )
   END_RUNG
   RUNG wire#w2
      Coil( "ST10Cylinder".Cy[39].In.GoHomeInterlock )
   END_RUNG
   RUNG wire#w1
      I_Contact( #AlwaysON )
      Coil( "ST10Cylinder".Cy[39].In.Error )
   END_RUNG
   // the same network as SCL:
   "ST10Cylinder".Cy[39].In.GoWorkInterlock := #AlwaysON AND #E_stop;
   "ST10Cylinder".Cy[39].In.GoHomeInterlock := #AlwaysON AND #E_stop;
   "ST10Cylinder".Cy[39].In.Error := #AlwaysON AND NOT #AlwaysON;
END_REGION

REGION Network 11: CY40 interface
   RUNG wire#powerrail
      Contact( #AlwaysON )
      wire#w1
      Contact( #E_stop )
      wire#w2
      Coil( "ST10Cylinder".Cy[40].In.GoWorkInterlock )
   END_RUNG
   RUNG wire#w2
      Coil( "ST10Cylinder".Cy[40].In.GoHomeInterlock )
   END_RUNG
   RUNG wire#w1
      I_Contact( #AlwaysON )
      Coil( "ST10Cylinder".Cy[40].In.Error )
   END_RUNG
   // the same network as SCL:
   "ST10Cylinder".Cy[40].In.GoWorkInterlock := #AlwaysON AND #E_stop;
   "ST10Cylinder".Cy[40].In.GoHomeInterlock := #AlwaysON AND #E_stop;
   "ST10Cylinder".Cy[40].In.Error := #AlwaysON AND NOT #AlwaysON;
END_REGION
END_FUNCTION

FUNCTION "ST10Cyl_interface41-50" : Void   // FC1024, LAD
{ S7_Optimized_Access := 'FALSE' }
// stored: AutoNumber false, SetENOAutomatically false
   VAR_INPUT
      AlwaysON : Bool;
      E_stop : Bool;
   END_VAR
   VAR_TEMP
      tTest : Bool;
   END_VAR
BEGIN

REGION Network 1 (SCL): Cylinder 41-50 IO Interface (SCL)
   //Cylinder41 IO  K-reserveLifting3LiftingCylinder
   //Input
   "ST10Cylinder".Cy[41].In.WorkPositionSensor := "iK-reserveLifting3LiftingCylinderInWP";
   "ST10Cylinder".Cy[41].In.HomePositionSensor := "iK-reserveLifting3LiftingCylinderInHP";
   //Output
   "oK-reserveLifting3LiftingCylinderToWP" := "ST10Cylinder".Cy[41].Out.GoWorkPosition;
   "oK-reserveLifting3LiftingCylinderToHP" := "ST10Cylinder".Cy[41].Out.GoHomePosition;

   //Cylinder42 IO  K-reserveLifting3PalletLocationCylinder
   //Input
   "ST10Cylinder".Cy[42].In.WorkPositionSensor := "iK-reserveLifting3PalletLocationCylinderInWP";
   "ST10Cylinder".Cy[42].In.HomePositionSensor := "iK-reserveLifting3PalletLocationCylinderInHP";
   //Output
   "oK-reserveLifting3PalletLocationCylinderToWP" := "ST10Cylinder".Cy[42].Out.GoWorkPosition;
   "oK-reserveLifting3PalletLocationCylinderToHP" := "ST10Cylinder".Cy[42].Out.GoHomePosition;

   //Cylinder43 IO  K-reserveLoadingStopperCylinder1
   //Input
   "ST10Cylinder".Cy[43].In.WorkPositionSensor := "oK-reserveLoadingStopperCylinder1_ToWP";
   "ST10Cylinder".Cy[43].In.HomePositionSensor := "oK-reserveLoadingStopperCylinder1_ToHP";
   //Output
   "oK-reserveLoadingStopperCylinder1_ToWP" := "ST10Cylinder".Cy[43].Out.GoWorkPosition;
   "oK-reserveLoadingStopperCylinder1_ToHP" := "ST10Cylinder".Cy[43].Out.GoHomePosition;

   //Cylinder44 IO  K-reserveLoadingStopperCylinder2
   //Input
   "ST10Cylinder".Cy[44].In.WorkPositionSensor := "oK-reserveLoadingStopperCylinder2_ToWP";
   "ST10Cylinder".Cy[44].In.HomePositionSensor := "oK-reserveLoadingStopperCylinder2_ToHP";
   //Output
   "oK-reserveLoadingStopperCylinder2_ToWP" := "ST10Cylinder".Cy[44].Out.GoWorkPosition;
   "oK-reserveLoadingStopperCylinder2_ToHP" := "ST10Cylinder".Cy[44].Out.GoHomePosition;

   //Cylinder45 IO  K-reserveLoadingStopperCylinder3
   //Input
   "ST10Cylinder".Cy[45].In.WorkPositionSensor := "oK-reserveLoadingStopperCylinder3_ToWP";
   "ST10Cylinder".Cy[45].In.HomePositionSensor := "oK-reserveLoadingStopperCylinder3_ToHP";
   //Output
   "oK-reserveLoadingStopperCylinder3_ToWP" := "ST10Cylinder".Cy[45].Out.GoWorkPosition;
   "oK-reserveLoadingStopperCylinder3_ToHP" := "ST10Cylinder".Cy[45].Out.GoHomePosition;

   //Cylinder46 K-reserveLoadingStopperCylinder4
   //Input
   "ST10Cylinder".Cy[46].In.WorkPositionSensor := "oK-reserveLoadingStopperCylinder4_ToWP";
   "ST10Cylinder".Cy[46].In.HomePositionSensor := "oK-reserveLoadingStopperCylinder4_ToHP";
   //Output
   "oK-reserveLoadingStopperCylinder4_ToWP" := "ST10Cylinder".Cy[46].Out.GoWorkPosition;
   "oK-reserveLoadingStopperCylinder4_ToHP" := "ST10Cylinder".Cy[46].Out.GoHomePosition;

   //Cylinder47 K-reserveTakeStopperCylinder1
   //Input
   "ST10Cylinder".Cy[47].In.WorkPositionSensor := "oK-reserveTakeStopperCylinder1_ToWP";
   "ST10Cylinder".Cy[47].In.HomePositionSensor := "oK-reserveTakeStopperCylinder1_ToHP";
   //Output
   "oK-reserveTakeStopperCylinder1_ToWP" := "ST10Cylinder".Cy[47].Out.GoWorkPosition;
   "oK-reserveTakeStopperCylinder1_ToHP" := "ST10Cylinder".Cy[47].Out.GoHomePosition;

   //Cylinder48 K-reserveTakeStopperCylinder2
   //Input
   "ST10Cylinder".Cy[48].In.WorkPositionSensor := "oK-reserveTakeStopperCylinder2_ToWP";
   "ST10Cylinder".Cy[48].In.HomePositionSensor := "oK-reserveTakeStopperCylinder2_ToHP";
   //Output
   "oK-reserveTakeStopperCylinder2_ToWP" := "ST10Cylinder".Cy[48].Out.GoWorkPosition;
   "oK-reserveTakeStopperCylinder2_ToHP" := "ST10Cylinder".Cy[48].Out.GoHomePosition;

   //Cylinder49 K-reserveTakeStopperCylinder3
   //Input
   "ST10Cylinder".Cy[49].In.WorkPositionSensor := "oK-reserveTakeStopperCylinder3_ToWP";
   "ST10Cylinder".Cy[49].In.HomePositionSensor := "oK-reserveTakeStopperCylinder3_ToHP";
   //Output
   "oK-reserveTakeStopperCylinder3_ToWP" := "ST10Cylinder".Cy[49].Out.GoWorkPosition;
   "oK-reserveTakeStopperCylinder3_ToHP" := "ST10Cylinder".Cy[49].Out.GoHomePosition;

   (*
   //Cylinder50 K-reserveLoadingStopperCylinder4_2
   // //Input
   "ST10Cylinder".Cy[50].In.WorkPositionSensor := "oK-reserveLoadingStopperCylinder4_2";
   "ST10Cylinder".Cy[50].In.HomePositionSensor := NOT "oK-reserveLoadingStopperCylinder4_2";
   // //Output
   "oK-reserveLoadingStopperCylinder4_2" := "ST10Cylinder".Cy[50].Out.GoWorkPosition;
   // "Feeding washer  lift Cylinder ToHP" := "ST10Cylinder".Cy[50].Out.GoHomePosition;
   *)
END_REGION

REGION Network 2: CY41 interface K-reserveLifting3LiftingCylinder
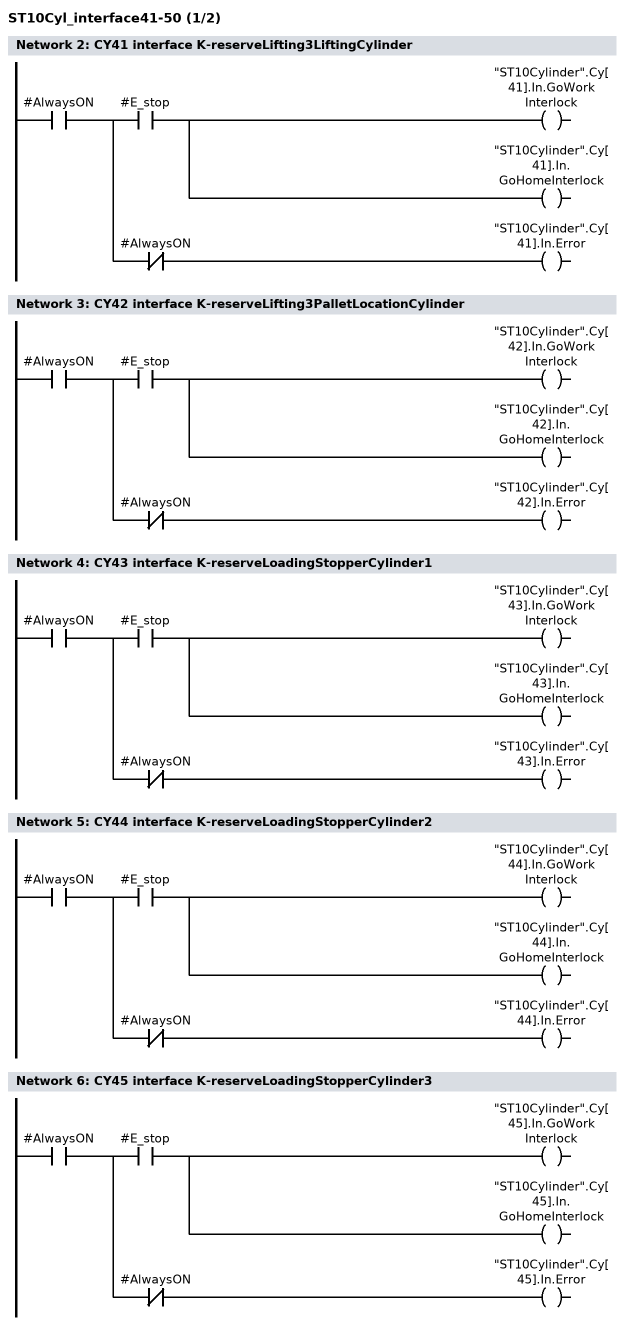
   RUNG wire#powerrail
      Contact( #AlwaysON )
      wire#w1
      Contact( #E_stop )
      wire#w2
      Coil( "ST10Cylinder".Cy[41].In.GoWorkInterlock )
   END_RUNG
   RUNG wire#w2
      Coil( "ST10Cylinder".Cy[41].In.GoHomeInterlock )
   END_RUNG
   RUNG wire#w1
      I_Contact( #AlwaysON )
      Coil( "ST10Cylinder".Cy[41].In.Error )
   END_RUNG
   // the same network as SCL:
   "ST10Cylinder".Cy[41].In.GoWorkInterlock := #AlwaysON AND #E_stop;
   "ST10Cylinder".Cy[41].In.GoHomeInterlock := #AlwaysON AND #E_stop;
   "ST10Cylinder".Cy[41].In.Error := #AlwaysON AND NOT #AlwaysON;
END_REGION

REGION Network 3: CY42 interface K-reserveLifting3PalletLocationCylinder
   RUNG wire#powerrail
      Contact( #AlwaysON )
      wire#w1
      Contact( #E_stop )
      wire#w2
      Coil( "ST10Cylinder".Cy[42].In.GoWorkInterlock )
   END_RUNG
   RUNG wire#w2
      Coil( "ST10Cylinder".Cy[42].In.GoHomeInterlock )
   END_RUNG
   RUNG wire#w1
      I_Contact( #AlwaysON )
      Coil( "ST10Cylinder".Cy[42].In.Error )
   END_RUNG
   // the same network as SCL:
   "ST10Cylinder".Cy[42].In.GoWorkInterlock := #AlwaysON AND #E_stop;
   "ST10Cylinder".Cy[42].In.GoHomeInterlock := #AlwaysON AND #E_stop;
   "ST10Cylinder".Cy[42].In.Error := #AlwaysON AND NOT #AlwaysON;
END_REGION

REGION Network 4: CY43 interface K-reserveLoadingStopperCylinder1
   RUNG wire#powerrail
      Contact( #AlwaysON )
      wire#w1
      Contact( #E_stop )
      wire#w2
      Coil( "ST10Cylinder".Cy[43].In.GoWorkInterlock )
   END_RUNG
   RUNG wire#w2
      Coil( "ST10Cylinder".Cy[43].In.GoHomeInterlock )
   END_RUNG
   RUNG wire#w1
      I_Contact( #AlwaysON )
      Coil( "ST10Cylinder".Cy[43].In.Error )
   END_RUNG
   // the same network as SCL:
   "ST10Cylinder".Cy[43].In.GoWorkInterlock := #AlwaysON AND #E_stop;
   "ST10Cylinder".Cy[43].In.GoHomeInterlock := #AlwaysON AND #E_stop;
   "ST10Cylinder".Cy[43].In.Error := #AlwaysON AND NOT #AlwaysON;
END_REGION

REGION Network 5: CY44 interface K-reserveLoadingStopperCylinder2
   RUNG wire#powerrail
      Contact( #AlwaysON )
      wire#w1
      Contact( #E_stop )
      wire#w2
      Coil( "ST10Cylinder".Cy[44].In.GoWorkInterlock )
   END_RUNG
   RUNG wire#w2
      Coil( "ST10Cylinder".Cy[44].In.GoHomeInterlock )
   END_RUNG
   RUNG wire#w1
      I_Contact( #AlwaysON )
      Coil( "ST10Cylinder".Cy[44].In.Error )
   END_RUNG
   // the same network as SCL:
   "ST10Cylinder".Cy[44].In.GoWorkInterlock := #AlwaysON AND #E_stop;
   "ST10Cylinder".Cy[44].In.GoHomeInterlock := #AlwaysON AND #E_stop;
   "ST10Cylinder".Cy[44].In.Error := #AlwaysON AND NOT #AlwaysON;
END_REGION

REGION Network 6: CY45 interface K-reserveLoadingStopperCylinder3
   RUNG wire#powerrail
      Contact( #AlwaysON )
      wire#w1
      Contact( #E_stop )
      wire#w2
      Coil( "ST10Cylinder".Cy[45].In.GoWorkInterlock )
   END_RUNG
   RUNG wire#w2
      Coil( "ST10Cylinder".Cy[45].In.GoHomeInterlock )
   END_RUNG
   RUNG wire#w1
      I_Contact( #AlwaysON )
      Coil( "ST10Cylinder".Cy[45].In.Error )
   END_RUNG
   // the same network as SCL:
   "ST10Cylinder".Cy[45].In.GoWorkInterlock := #AlwaysON AND #E_stop;
   "ST10Cylinder".Cy[45].In.GoHomeInterlock := #AlwaysON AND #E_stop;
   "ST10Cylinder".Cy[45].In.Error := #AlwaysON AND NOT #AlwaysON;
END_REGION

REGION Network 7: CY46 interface K-reserveLoadingStopperCylinder4
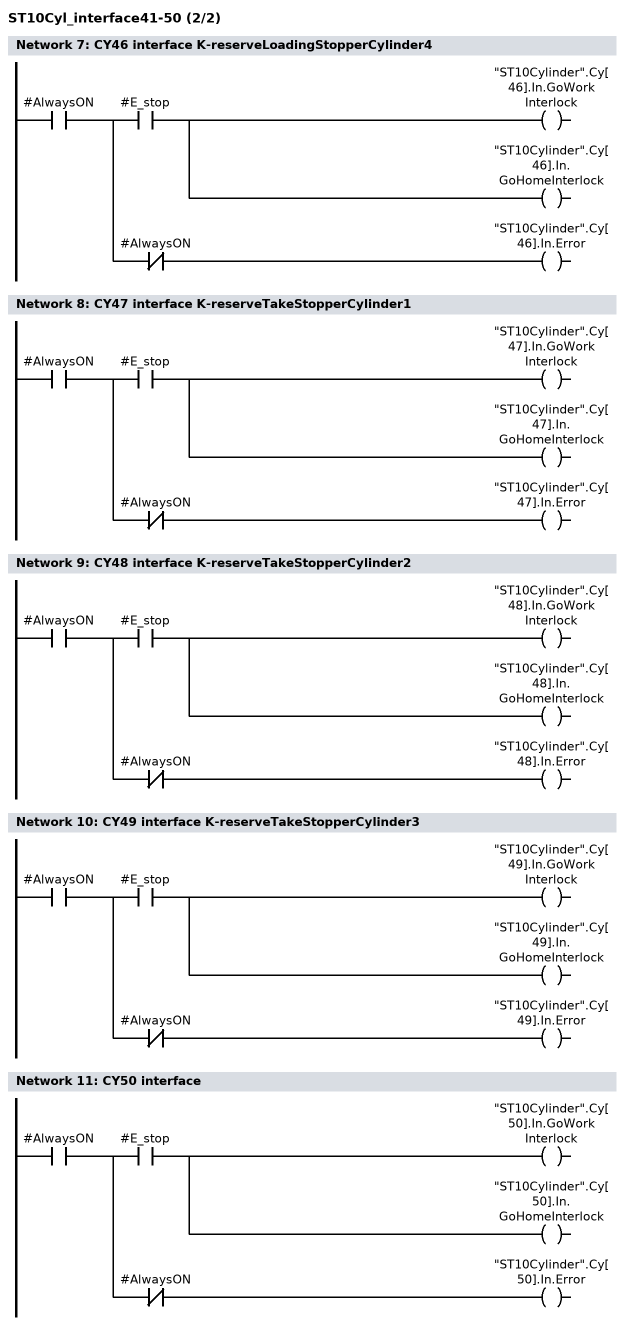
   RUNG wire#powerrail
      Contact( #AlwaysON )
      wire#w1
      Contact( #E_stop )
      wire#w2
      Coil( "ST10Cylinder".Cy[46].In.GoWorkInterlock )
   END_RUNG
   RUNG wire#w2
      Coil( "ST10Cylinder".Cy[46].In.GoHomeInterlock )
   END_RUNG
   RUNG wire#w1
      I_Contact( #AlwaysON )
      Coil( "ST10Cylinder".Cy[46].In.Error )
   END_RUNG
   // the same network as SCL:
   "ST10Cylinder".Cy[46].In.GoWorkInterlock := #AlwaysON AND #E_stop;
   "ST10Cylinder".Cy[46].In.GoHomeInterlock := #AlwaysON AND #E_stop;
   "ST10Cylinder".Cy[46].In.Error := #AlwaysON AND NOT #AlwaysON;
END_REGION

REGION Network 8: CY47 interface K-reserveTakeStopperCylinder1
   RUNG wire#powerrail
      Contact( #AlwaysON )
      wire#w1
      Contact( #E_stop )
      wire#w2
      Coil( "ST10Cylinder".Cy[47].In.GoWorkInterlock )
   END_RUNG
   RUNG wire#w2
      Coil( "ST10Cylinder".Cy[47].In.GoHomeInterlock )
   END_RUNG
   RUNG wire#w1
      I_Contact( #AlwaysON )
      Coil( "ST10Cylinder".Cy[47].In.Error )
   END_RUNG
   // the same network as SCL:
   "ST10Cylinder".Cy[47].In.GoWorkInterlock := #AlwaysON AND #E_stop;
   "ST10Cylinder".Cy[47].In.GoHomeInterlock := #AlwaysON AND #E_stop;
   "ST10Cylinder".Cy[47].In.Error := #AlwaysON AND NOT #AlwaysON;
END_REGION

REGION Network 9: CY48 interface K-reserveTakeStopperCylinder2
   RUNG wire#powerrail
      Contact( #AlwaysON )
      wire#w1
      Contact( #E_stop )
      wire#w2
      Coil( "ST10Cylinder".Cy[48].In.GoWorkInterlock )
   END_RUNG
   RUNG wire#w2
      Coil( "ST10Cylinder".Cy[48].In.GoHomeInterlock )
   END_RUNG
   RUNG wire#w1
      I_Contact( #AlwaysON )
      Coil( "ST10Cylinder".Cy[48].In.Error )
   END_RUNG
   // the same network as SCL:
   "ST10Cylinder".Cy[48].In.GoWorkInterlock := #AlwaysON AND #E_stop;
   "ST10Cylinder".Cy[48].In.GoHomeInterlock := #AlwaysON AND #E_stop;
   "ST10Cylinder".Cy[48].In.Error := #AlwaysON AND NOT #AlwaysON;
END_REGION

REGION Network 10: CY49 interface K-reserveTakeStopperCylinder3
   RUNG wire#powerrail
      Contact( #AlwaysON )
      wire#w1
      Contact( #E_stop )
      wire#w2
      Coil( "ST10Cylinder".Cy[49].In.GoWorkInterlock )
   END_RUNG
   RUNG wire#w2
      Coil( "ST10Cylinder".Cy[49].In.GoHomeInterlock )
   END_RUNG
   RUNG wire#w1
      I_Contact( #AlwaysON )
      Coil( "ST10Cylinder".Cy[49].In.Error )
   END_RUNG
   // the same network as SCL:
   "ST10Cylinder".Cy[49].In.GoWorkInterlock := #AlwaysON AND #E_stop;
   "ST10Cylinder".Cy[49].In.GoHomeInterlock := #AlwaysON AND #E_stop;
   "ST10Cylinder".Cy[49].In.Error := #AlwaysON AND NOT #AlwaysON;
END_REGION

REGION Network 11: CY50 interface
   RUNG wire#powerrail
      Contact( #AlwaysON )
      wire#w1
      Contact( #E_stop )
      wire#w2
      Coil( "ST10Cylinder".Cy[50].In.GoWorkInterlock )
   END_RUNG
   RUNG wire#w2
      Coil( "ST10Cylinder".Cy[50].In.GoHomeInterlock )
   END_RUNG
   RUNG wire#w1
      I_Contact( #AlwaysON )
      Coil( "ST10Cylinder".Cy[50].In.Error )
   END_RUNG
   // the same network as SCL:
   "ST10Cylinder".Cy[50].In.GoWorkInterlock := #AlwaysON AND #E_stop;
   "ST10Cylinder".Cy[50].In.GoHomeInterlock := #AlwaysON AND #E_stop;
   "ST10Cylinder".Cy[50].In.Error := #AlwaysON AND NOT #AlwaysON;
END_REGION
END_FUNCTION

FUNCTION "ST10Cyl_interface51-60" : Void   // FC1025, LAD
{ S7_Optimized_Access := 'FALSE' }
// stored: AutoNumber false, SetENOAutomatically false
   VAR_INPUT
      AlwaysON : Bool;
      E_stop : Bool;
   END_VAR
   VAR_TEMP
      tTest : Bool;
   END_VAR
   VAR_TEMP   // added for the SCL form of the ladder/FBD networks
      _w1 : Bool;
   END_VAR
BEGIN

REGION Network 1 (SCL): Cylinder 51-60 IO Interface (SCL)

   //Cylinder51 IO  L-UnloadingTransCylinder
   //Input
   "ST10Cylinder".Cy[51].In.WorkPositionSensor := "iL-UnloadingTransCylinderInWP";
   "ST10Cylinder".Cy[51].In.HomePositionSensor := "iL-UnloadingTransCylinderInHP";
   //Output
   "oL-UnloadingTransCylinderToWP" := "ST10Cylinder".Cy[51].Out.GoWorkPosition;
   "oL-UnloadingTransCylinderToHP" := "ST10Cylinder".Cy[51].Out.GoHomePosition;

   //Cylinder52 IO  L-UnloadingTransPalletLocationCylinder
   //Input
   "ST10Cylinder".Cy[52].In.WorkPositionSensor := "iL-UnloadingTransPalletLocationCylinderInWP";
   "ST10Cylinder".Cy[52].In.HomePositionSensor := "iL-UnloadingTransPalletLocationCylinderInHP";
   //Output
   "oL-UnloadingTransPalletLocationCylinderToWP" := "ST10Cylinder".Cy[52].Out.GoWorkPosition;
   "oL-UnloadingTransPalletLocationCylinderToHP" := "ST10Cylinder".Cy[52].Out.GoHomePosition;

   //Cylinder53 IO  L-UnloadingStopperCylinder1
   //Input
   "ST10Cylinder".Cy[53].In.WorkPositionSensor := "oL-UnloadingStopperCylinder1_ToWP";
   "ST10Cylinder".Cy[53].In.HomePositionSensor := "oL-UnloadingStopperCylinder1_ToHP";
   //Output
   "oL-UnloadingStopperCylinder1_ToWP" := "ST10Cylinder".Cy[53].Out.GoWorkPosition;
   "oL-UnloadingStopperCylinder1_ToHP" := "ST10Cylinder".Cy[53].Out.GoHomePosition;

   //Cylinder54 IO  L-UnloadingStopperCylinder2
   //Input
   "ST10Cylinder".Cy[54].In.WorkPositionSensor := "oL-UnloadingStopperCylinder2_ToWP";
   "ST10Cylinder".Cy[54].In.HomePositionSensor := "oL-UnloadingStopperCylinder2_ToHP";
   //Output
   "oL-UnloadingStopperCylinder2_ToWP" := "ST10Cylinder".Cy[54].Out.GoWorkPosition;
   "oL-UnloadingStopperCylinder2_ToHP" := "ST10Cylinder".Cy[54].Out.GoHomePosition;

   //Cylinder55 IO  L-UnloadingStopperCylinder3
   //Input
   "ST10Cylinder".Cy[55].In.WorkPositionSensor := "oL-UnloadingStopperCylinder3_ToWP";
   "ST10Cylinder".Cy[55].In.HomePositionSensor := "oL-UnloadingStopperCylinder3_ToHP";
   //Output
   "oL-UnloadingStopperCylinder3_ToWP" := "ST10Cylinder".Cy[55].Out.GoWorkPosition;
   "oL-UnloadingStopperCylinder3_ToHP" := "ST10Cylinder".Cy[55].Out.GoHomePosition;

   (*
   //Cylinder56  L-UnloadingStopperCylinder2_2
   //Input
   "ST10Cylinder".Cy[56].In.WorkPositionSensor := "oL-UnloadingStopperCylinder2_2";
   "ST10Cylinder".Cy[56].In.HomePositionSensor := NOT "oL-UnloadingStopperCylinder2_2";
   //Output
   "oL-UnloadingStopperCylinder2_2" := "ST10Cylinder".Cy[56].Out.GoWorkPosition;
   //"oI-0080TrayLoadingTraySupportCylinder1ToHP" := "ST10Cylinder".Cy[56].Out.GoHomePosition;

   //Cylinder57 L-UnloadingStopperCylinder3_1
   //Input
   "ST10Cylinder".Cy[57].In.WorkPositionSensor := "oL-UnloadingStopperCylinder3_1";
   "ST10Cylinder".Cy[57].In.HomePositionSensor := NOT "oL-UnloadingStopperCylinder3_1";
   //Output
   "oL-UnloadingStopperCylinder3_1" := "ST10Cylinder".Cy[57].Out.GoWorkPosition;
   //"oI-0070TrayLoadingTraySupportCylinder8ToHP" := "ST10Cylinder".Cy[57].Out.GoHomePosition;

   //Cylinder58 L-UnloadingStopperCylinder3_2
   //Input
   "ST10Cylinder".Cy[58].In.WorkPositionSensor := "oL-UnloadingStopperCylinder3_2";
   "ST10Cylinder".Cy[58].In.HomePositionSensor := NOT "oL-UnloadingStopperCylinder3_2";
   //Output
   "oL-UnloadingStopperCylinder3_2" := "ST10Cylinder".Cy[58].Out.GoWorkPosition;
   //"oI-0080TrayLoadingTrayLocationCylinderToHP" := "ST10Cylinder".Cy[58].Out.GoHomePosition;
   //

   *)
END_REGION

REGION Network 2: CY51 interface L-UnloadingTransCylinder
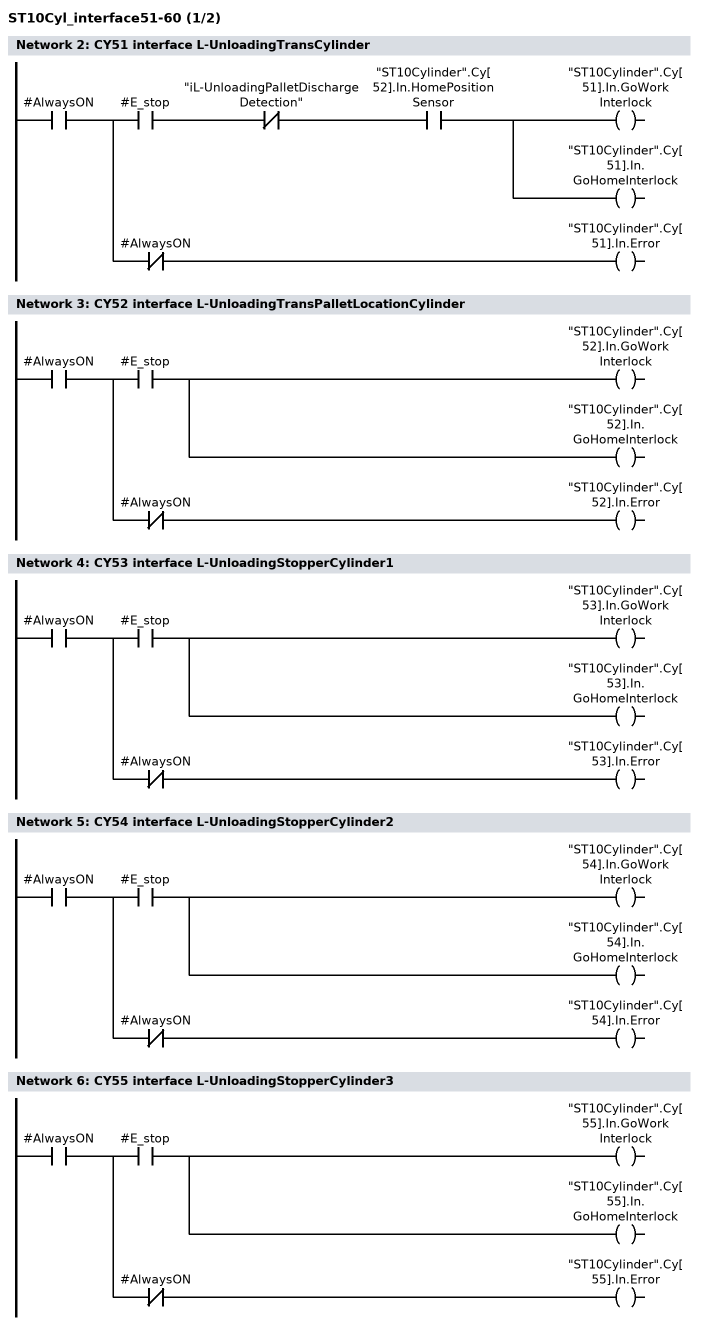
   RUNG wire#powerrail
      Contact( #AlwaysON )
      wire#w1
      Contact( #E_stop )
      I_Contact( "iL-UnloadingPalletDischargeDetection" )
      Contact( "ST10Cylinder".Cy[52].In.HomePositionSensor )
      wire#w2
      Coil( "ST10Cylinder".Cy[51].In.GoWorkInterlock )
   END_RUNG
   RUNG wire#w2
      Coil( "ST10Cylinder".Cy[51].In.GoHomeInterlock )
   END_RUNG
   RUNG wire#w1
      I_Contact( #AlwaysON )
      Coil( "ST10Cylinder".Cy[51].In.Error )
   END_RUNG
   // the same network as SCL:
   #_w1 := #AlwaysON AND #E_stop AND NOT "iL-UnloadingPalletDischargeDetection" AND "ST10Cylinder".Cy[52].In.HomePositionSensor;
   "ST10Cylinder".Cy[51].In.GoWorkInterlock := #AlwaysON AND #E_stop AND NOT "iL-UnloadingPalletDischargeDetection" AND "ST10Cylinder".Cy[52].In.HomePositionSensor;
   "ST10Cylinder".Cy[51].In.GoHomeInterlock := #_w1;
   "ST10Cylinder".Cy[51].In.Error := #AlwaysON AND NOT #AlwaysON;
END_REGION

REGION Network 3: CY52 interface L-UnloadingTransPalletLocationCylinder
   RUNG wire#powerrail
      Contact( #AlwaysON )
      wire#w1
      Contact( #E_stop )
      wire#w2
      Coil( "ST10Cylinder".Cy[52].In.GoWorkInterlock )
   END_RUNG
   RUNG wire#w2
      Coil( "ST10Cylinder".Cy[52].In.GoHomeInterlock )
   END_RUNG
   RUNG wire#w1
      I_Contact( #AlwaysON )
      Coil( "ST10Cylinder".Cy[52].In.Error )
   END_RUNG
   // the same network as SCL:
   "ST10Cylinder".Cy[52].In.GoWorkInterlock := #AlwaysON AND #E_stop;
   "ST10Cylinder".Cy[52].In.GoHomeInterlock := #AlwaysON AND #E_stop;
   "ST10Cylinder".Cy[52].In.Error := #AlwaysON AND NOT #AlwaysON;
END_REGION

REGION Network 4: CY53 interface L-UnloadingStopperCylinder1
   RUNG wire#powerrail
      Contact( #AlwaysON )
      wire#w1
      Contact( #E_stop )
      wire#w2
      Coil( "ST10Cylinder".Cy[53].In.GoWorkInterlock )
   END_RUNG
   RUNG wire#w2
      Coil( "ST10Cylinder".Cy[53].In.GoHomeInterlock )
   END_RUNG
   RUNG wire#w1
      I_Contact( #AlwaysON )
      Coil( "ST10Cylinder".Cy[53].In.Error )
   END_RUNG
   // the same network as SCL:
   "ST10Cylinder".Cy[53].In.GoWorkInterlock := #AlwaysON AND #E_stop;
   "ST10Cylinder".Cy[53].In.GoHomeInterlock := #AlwaysON AND #E_stop;
   "ST10Cylinder".Cy[53].In.Error := #AlwaysON AND NOT #AlwaysON;
END_REGION

REGION Network 5: CY54 interface L-UnloadingStopperCylinder2
   RUNG wire#powerrail
      Contact( #AlwaysON )
      wire#w1
      Contact( #E_stop )
      wire#w2
      Coil( "ST10Cylinder".Cy[54].In.GoWorkInterlock )
   END_RUNG
   RUNG wire#w2
      Coil( "ST10Cylinder".Cy[54].In.GoHomeInterlock )
   END_RUNG
   RUNG wire#w1
      I_Contact( #AlwaysON )
      Coil( "ST10Cylinder".Cy[54].In.Error )
   END_RUNG
   // the same network as SCL:
   "ST10Cylinder".Cy[54].In.GoWorkInterlock := #AlwaysON AND #E_stop;
   "ST10Cylinder".Cy[54].In.GoHomeInterlock := #AlwaysON AND #E_stop;
   "ST10Cylinder".Cy[54].In.Error := #AlwaysON AND NOT #AlwaysON;
END_REGION

REGION Network 6: CY55 interface L-UnloadingStopperCylinder3
   RUNG wire#powerrail
      Contact( #AlwaysON )
      wire#w1
      Contact( #E_stop )
      wire#w2
      Coil( "ST10Cylinder".Cy[55].In.GoWorkInterlock )
   END_RUNG
   RUNG wire#w2
      Coil( "ST10Cylinder".Cy[55].In.GoHomeInterlock )
   END_RUNG
   RUNG wire#w1
      I_Contact( #AlwaysON )
      Coil( "ST10Cylinder".Cy[55].In.Error )
   END_RUNG
   // the same network as SCL:
   "ST10Cylinder".Cy[55].In.GoWorkInterlock := #AlwaysON AND #E_stop;
   "ST10Cylinder".Cy[55].In.GoHomeInterlock := #AlwaysON AND #E_stop;
   "ST10Cylinder".Cy[55].In.Error := #AlwaysON AND NOT #AlwaysON;
END_REGION

REGION Network 7: CY56 interface
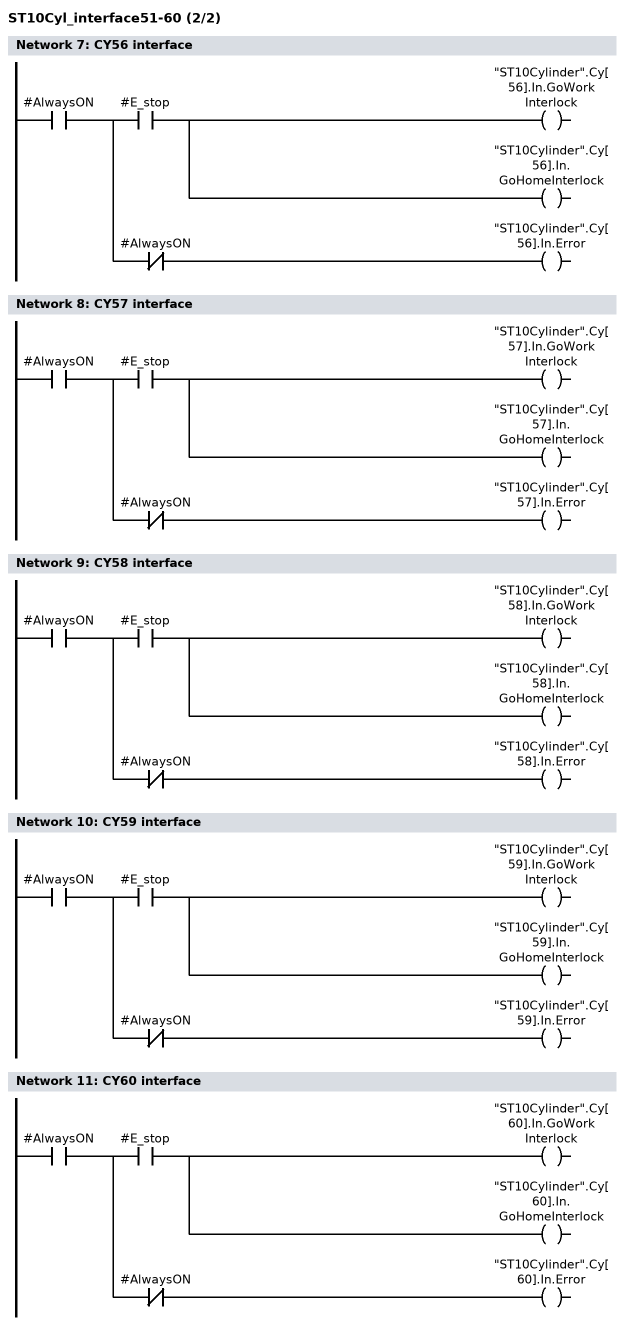
   RUNG wire#powerrail
      Contact( #AlwaysON )
      wire#w1
      Contact( #E_stop )
      wire#w2
      Coil( "ST10Cylinder".Cy[56].In.GoWorkInterlock )
   END_RUNG
   RUNG wire#w2
      Coil( "ST10Cylinder".Cy[56].In.GoHomeInterlock )
   END_RUNG
   RUNG wire#w1
      I_Contact( #AlwaysON )
      Coil( "ST10Cylinder".Cy[56].In.Error )
   END_RUNG
   // the same network as SCL:
   "ST10Cylinder".Cy[56].In.GoWorkInterlock := #AlwaysON AND #E_stop;
   "ST10Cylinder".Cy[56].In.GoHomeInterlock := #AlwaysON AND #E_stop;
   "ST10Cylinder".Cy[56].In.Error := #AlwaysON AND NOT #AlwaysON;
END_REGION

REGION Network 8: CY57 interface
   RUNG wire#powerrail
      Contact( #AlwaysON )
      wire#w1
      Contact( #E_stop )
      wire#w2
      Coil( "ST10Cylinder".Cy[57].In.GoWorkInterlock )
   END_RUNG
   RUNG wire#w2
      Coil( "ST10Cylinder".Cy[57].In.GoHomeInterlock )
   END_RUNG
   RUNG wire#w1
      I_Contact( #AlwaysON )
      Coil( "ST10Cylinder".Cy[57].In.Error )
   END_RUNG
   // the same network as SCL:
   "ST10Cylinder".Cy[57].In.GoWorkInterlock := #AlwaysON AND #E_stop;
   "ST10Cylinder".Cy[57].In.GoHomeInterlock := #AlwaysON AND #E_stop;
   "ST10Cylinder".Cy[57].In.Error := #AlwaysON AND NOT #AlwaysON;
END_REGION

REGION Network 9: CY58 interface
   RUNG wire#powerrail
      Contact( #AlwaysON )
      wire#w1
      Contact( #E_stop )
      wire#w2
      Coil( "ST10Cylinder".Cy[58].In.GoWorkInterlock )
   END_RUNG
   RUNG wire#w2
      Coil( "ST10Cylinder".Cy[58].In.GoHomeInterlock )
   END_RUNG
   RUNG wire#w1
      I_Contact( #AlwaysON )
      Coil( "ST10Cylinder".Cy[58].In.Error )
   END_RUNG
   // the same network as SCL:
   "ST10Cylinder".Cy[58].In.GoWorkInterlock := #AlwaysON AND #E_stop;
   "ST10Cylinder".Cy[58].In.GoHomeInterlock := #AlwaysON AND #E_stop;
   "ST10Cylinder".Cy[58].In.Error := #AlwaysON AND NOT #AlwaysON;
END_REGION

REGION Network 10: CY59 interface
   RUNG wire#powerrail
      Contact( #AlwaysON )
      wire#w1
      Contact( #E_stop )
      wire#w2
      Coil( "ST10Cylinder".Cy[59].In.GoWorkInterlock )
   END_RUNG
   RUNG wire#w2
      Coil( "ST10Cylinder".Cy[59].In.GoHomeInterlock )
   END_RUNG
   RUNG wire#w1
      I_Contact( #AlwaysON )
      Coil( "ST10Cylinder".Cy[59].In.Error )
   END_RUNG
   // the same network as SCL:
   "ST10Cylinder".Cy[59].In.GoWorkInterlock := #AlwaysON AND #E_stop;
   "ST10Cylinder".Cy[59].In.GoHomeInterlock := #AlwaysON AND #E_stop;
   "ST10Cylinder".Cy[59].In.Error := #AlwaysON AND NOT #AlwaysON;
END_REGION

REGION Network 11: CY60 interface
   RUNG wire#powerrail
      Contact( #AlwaysON )
      wire#w1
      Contact( #E_stop )
      wire#w2
      Coil( "ST10Cylinder".Cy[60].In.GoWorkInterlock )
   END_RUNG
   RUNG wire#w2
      Coil( "ST10Cylinder".Cy[60].In.GoHomeInterlock )
   END_RUNG
   RUNG wire#w1
      I_Contact( #AlwaysON )
      Coil( "ST10Cylinder".Cy[60].In.Error )
   END_RUNG
   // the same network as SCL:
   "ST10Cylinder".Cy[60].In.GoWorkInterlock := #AlwaysON AND #E_stop;
   "ST10Cylinder".Cy[60].In.GoHomeInterlock := #AlwaysON AND #E_stop;
   "ST10Cylinder".Cy[60].In.Error := #AlwaysON AND NOT #AlwaysON;
END_REGION
END_FUNCTION

FUNCTION "ST10Cyl_interface61-70" : Void   // FC1026, LAD
{ S7_Optimized_Access := 'FALSE' }
// stored: AutoNumber false, SetENOAutomatically false
   VAR_INPUT
      AlwaysON : Bool;
      E_stop : Bool;
   END_VAR
   VAR_TEMP
      tTest : Bool;
   END_VAR
BEGIN

REGION Network 1 (SCL): Cylinder 61-70 IO Interface (SCL)
   (*
   //Cylinder61 IO  K-reserveLifting3LiftingCylinder
   //Input
   "ST10Cylinder".Cy[61].In.WorkPositionSensor := "iK-reserveLifting3LiftingCylinderInWP";
   "ST10Cylinder".Cy[61].In.HomePositionSensor := "iK-reserveLifting3LiftingCylinderInHP";
   //Output
   "oK-reserveLifting3LiftingCylinderToWP" := "ST10Cylinder".Cy[61].Out.GoWorkPosition;
   "oK-reserveLifting3LiftingCylinderToHP" := "ST10Cylinder".Cy[61].Out.GoHomePosition;

   //Cylinder62 IO  K-reserveLifting3PalletLocationCylinder
   //Input
   "ST10Cylinder".Cy[62].In.WorkPositionSensor := "iK-reserveLifting3PalletLocationCylinderInWP";
   "ST10Cylinder".Cy[62].In.HomePositionSensor := "iK-reserveLifting3PalletLocationCylinderInHP";
   //Output
   "oK-reserveLifting3PalletLocationCylinderToWP" := "ST10Cylinder".Cy[62].Out.GoWorkPosition;
   "oK-reserveLifting3PalletLocationCylinderToHP" := "ST10Cylinder".Cy[62].Out.GoHomePosition;

   //Cylinder63 IO  K-reserveLoadingStopperCylinder1_1
   //Input
   "ST10Cylinder".Cy[63].In.WorkPositionSensor := "oK-reserveLoadingStopperCylinder1_1";
   "ST10Cylinder".Cy[63].In.HomePositionSensor := NOT "oK-reserveLoadingStopperCylinder1_1";
   //Output
   "oK-reserveLoadingStopperCylinder1_1" := "ST10Cylinder".Cy[63].Out.GoWorkPosition;
   //"oI-0030TrayLoading6trayStopperCylinderToHP" := "ST10Cylinder".Cy[63].Out.GoHomePosition;

   //Cylinder64 IO  K-reserveLoadingStopperCylinder1_2
   //Input
   "ST10Cylinder".Cy[64].In.WorkPositionSensor := "oK-reserveLoadingStopperCylinder1_2";
   "ST10Cylinder".Cy[64].In.HomePositionSensor := NOT "oK-reserveLoadingStopperCylinder1_2";
   //Output
   "oK-reserveLoadingStopperCylinder1_2" := "ST10Cylinder".Cy[64].Out.GoWorkPosition;
   //"oI-0060TrayLoadingTaketrayCylinderToHP" := "ST10Cylinder".Cy[64].Out.GoHomePosition;

   //Cylinder65 IO  K-reserveLoadingStopperCylinder2_1
   //Input
   "ST10Cylinder".Cy[65].In.WorkPositionSensor := "oK-reserveLoadingStopperCylinder2_1";
   "ST10Cylinder".Cy[65].In.HomePositionSensor := NOT "oK-reserveLoadingStopperCylinder2_1";
   //Output
   "oK-reserveLoadingStopperCylinder2_1" := "ST10Cylinder".Cy[65].Out.GoWorkPosition;
   //"oI-0050TrayLoadingTrayCylinderToHP" := "ST10Cylinder".Cy[65].Out.GoHomePosition;

   //Cylinder66 K-reserveLoadingStopperCylinder2_2
   //Input
   "ST10Cylinder".Cy[66].In.WorkPositionSensor := "oK-reserveLoadingStopperCylinder2_2";
   "ST10Cylinder".Cy[66].In.HomePositionSensor := NOT "oK-reserveLoadingStopperCylinder2_2";
   //Output
   "oK-reserveLoadingStopperCylinder2_2" := "ST10Cylinder".Cy[66].Out.GoWorkPosition;
   //"oI-0060TrayLoadingTraySupportCylinder1ToHP" := "ST10Cylinder".Cy[66].Out.GoHomePosition;

   //Cylinder67 K-reserveLoadingStopperCylinder3_1
   //Input
   "ST10Cylinder".Cy[67].In.WorkPositionSensor := "oK-reserveLoadingStopperCylinder3_1";
   "ST10Cylinder".Cy[67].In.HomePositionSensor := NOT "oK-reserveLoadingStopperCylinder3_1";
   //Output
   "oK-reserveLoadingStopperCylinder3_1" := "ST10Cylinder".Cy[67].Out.GoWorkPosition;
   //"oI-0070TrayLoadingTraySupportCylinder6ToHP" := "ST10Cylinder".Cy[67].Out.GoHomePosition;

   //Cylinder68 K-reserveLoadingStopperCylinder3_2
   //Input
   "ST10Cylinder".Cy[68].In.WorkPositionSensor := "oK-reserveLoadingStopperCylinder3_2";
   "ST10Cylinder".Cy[68].In.HomePositionSensor := NOT "oK-reserveLoadingStopperCylinder3_2";
   //Output
   "oK-reserveLoadingStopperCylinder3_2" := "ST10Cylinder".Cy[68].Out.GoWorkPosition;
   //"oI-0080TrayLoadingTrayLocationCylinderToHP" := "ST10Cylinder".Cy[68].Out.GoHomePosition;

   //Cylinder69 K-reserveLoadingStopperCylinder4_1
   //Input
   "ST10Cylinder".Cy[69].In.WorkPositionSensor := "oK-reserveLoadingStopperCylinder4_1";
   "ST10Cylinder".Cy[69].In.HomePositionSensor := NOT "oK-reserveLoadingStopperCylinder4_1";
   //Output
   "oK-reserveLoadingStopperCylinder4_1" := "ST10Cylinder".Cy[69].Out.GoWorkPosition;
   //"oI-0090TrayLoadingTrayUnloadingLiftingCylinderToHP" := "ST10Cylinder".Cy[69].Out.GoHomePosition;

   //Cylinder70 K-reserveLoadingStopperCylinder4_2
   // //Input
   "ST10Cylinder".Cy[70].In.WorkPositionSensor := "oK-reserveLoadingStopperCylinder4_2";
   "ST10Cylinder".Cy[70].In.HomePositionSensor := NOT "oK-reserveLoadingStopperCylinder4_2";
   // //Output
   "oK-reserveLoadingStopperCylinder4_2" := "ST10Cylinder".Cy[70].Out.GoWorkPosition;
   // "Feeding washer  lift Cylinder ToHP" := "ST10Cylinder".Cy[70].Out.GoHomePosition;
   *)
END_REGION

REGION Network 2: CY61 interface K-reserveLifting3LiftingCylinder
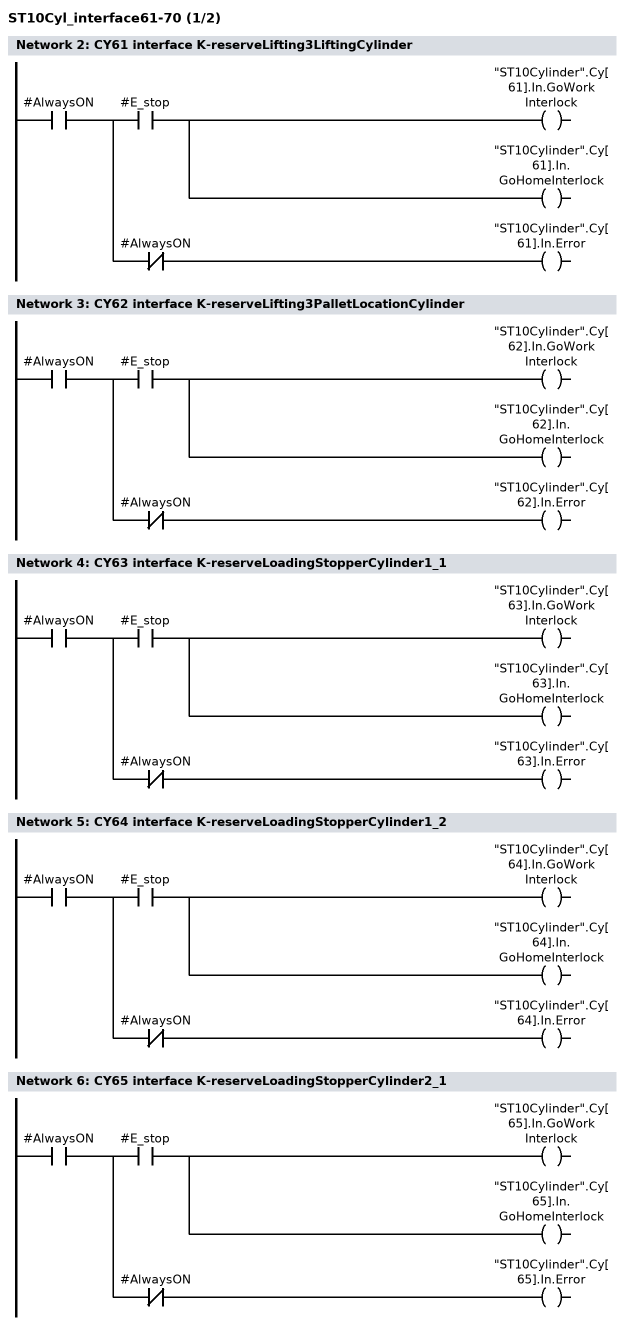
   RUNG wire#powerrail
      Contact( #AlwaysON )
      wire#w1
      Contact( #E_stop )
      wire#w2
      Coil( "ST10Cylinder".Cy[61].In.GoWorkInterlock )
   END_RUNG
   RUNG wire#w2
      Coil( "ST10Cylinder".Cy[61].In.GoHomeInterlock )
   END_RUNG
   RUNG wire#w1
      I_Contact( #AlwaysON )
      Coil( "ST10Cylinder".Cy[61].In.Error )
   END_RUNG
   // the same network as SCL:
   "ST10Cylinder".Cy[61].In.GoWorkInterlock := #AlwaysON AND #E_stop;
   "ST10Cylinder".Cy[61].In.GoHomeInterlock := #AlwaysON AND #E_stop;
   "ST10Cylinder".Cy[61].In.Error := #AlwaysON AND NOT #AlwaysON;
END_REGION

REGION Network 3: CY62 interface K-reserveLifting3PalletLocationCylinder
   RUNG wire#powerrail
      Contact( #AlwaysON )
      wire#w1
      Contact( #E_stop )
      wire#w2
      Coil( "ST10Cylinder".Cy[62].In.GoWorkInterlock )
   END_RUNG
   RUNG wire#w2
      Coil( "ST10Cylinder".Cy[62].In.GoHomeInterlock )
   END_RUNG
   RUNG wire#w1
      I_Contact( #AlwaysON )
      Coil( "ST10Cylinder".Cy[62].In.Error )
   END_RUNG
   // the same network as SCL:
   "ST10Cylinder".Cy[62].In.GoWorkInterlock := #AlwaysON AND #E_stop;
   "ST10Cylinder".Cy[62].In.GoHomeInterlock := #AlwaysON AND #E_stop;
   "ST10Cylinder".Cy[62].In.Error := #AlwaysON AND NOT #AlwaysON;
END_REGION

REGION Network 4: CY63 interface K-reserveLoadingStopperCylinder1_1
   RUNG wire#powerrail
      Contact( #AlwaysON )
      wire#w1
      Contact( #E_stop )
      wire#w2
      Coil( "ST10Cylinder".Cy[63].In.GoWorkInterlock )
   END_RUNG
   RUNG wire#w2
      Coil( "ST10Cylinder".Cy[63].In.GoHomeInterlock )
   END_RUNG
   RUNG wire#w1
      I_Contact( #AlwaysON )
      Coil( "ST10Cylinder".Cy[63].In.Error )
   END_RUNG
   // the same network as SCL:
   "ST10Cylinder".Cy[63].In.GoWorkInterlock := #AlwaysON AND #E_stop;
   "ST10Cylinder".Cy[63].In.GoHomeInterlock := #AlwaysON AND #E_stop;
   "ST10Cylinder".Cy[63].In.Error := #AlwaysON AND NOT #AlwaysON;
END_REGION

REGION Network 5: CY64 interface K-reserveLoadingStopperCylinder1_2
   RUNG wire#powerrail
      Contact( #AlwaysON )
      wire#w1
      Contact( #E_stop )
      wire#w2
      Coil( "ST10Cylinder".Cy[64].In.GoWorkInterlock )
   END_RUNG
   RUNG wire#w2
      Coil( "ST10Cylinder".Cy[64].In.GoHomeInterlock )
   END_RUNG
   RUNG wire#w1
      I_Contact( #AlwaysON )
      Coil( "ST10Cylinder".Cy[64].In.Error )
   END_RUNG
   // the same network as SCL:
   "ST10Cylinder".Cy[64].In.GoWorkInterlock := #AlwaysON AND #E_stop;
   "ST10Cylinder".Cy[64].In.GoHomeInterlock := #AlwaysON AND #E_stop;
   "ST10Cylinder".Cy[64].In.Error := #AlwaysON AND NOT #AlwaysON;
END_REGION

REGION Network 6: CY65 interface K-reserveLoadingStopperCylinder2_1
   RUNG wire#powerrail
      Contact( #AlwaysON )
      wire#w1
      Contact( #E_stop )
      wire#w2
      Coil( "ST10Cylinder".Cy[65].In.GoWorkInterlock )
   END_RUNG
   RUNG wire#w2
      Coil( "ST10Cylinder".Cy[65].In.GoHomeInterlock )
   END_RUNG
   RUNG wire#w1
      I_Contact( #AlwaysON )
      Coil( "ST10Cylinder".Cy[65].In.Error )
   END_RUNG
   // the same network as SCL:
   "ST10Cylinder".Cy[65].In.GoWorkInterlock := #AlwaysON AND #E_stop;
   "ST10Cylinder".Cy[65].In.GoHomeInterlock := #AlwaysON AND #E_stop;
   "ST10Cylinder".Cy[65].In.Error := #AlwaysON AND NOT #AlwaysON;
END_REGION

REGION Network 7: CY66 interface K-reserveLoadingStopperCylinder2_2
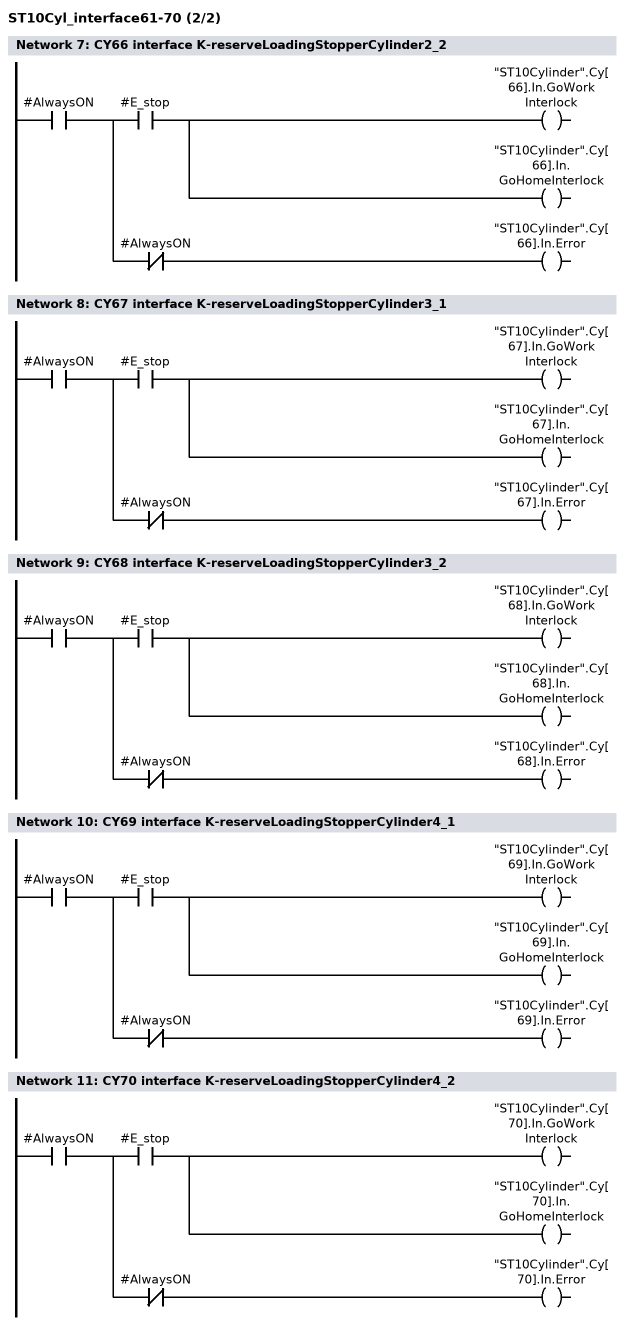
   RUNG wire#powerrail
      Contact( #AlwaysON )
      wire#w1
      Contact( #E_stop )
      wire#w2
      Coil( "ST10Cylinder".Cy[66].In.GoWorkInterlock )
   END_RUNG
   RUNG wire#w2
      Coil( "ST10Cylinder".Cy[66].In.GoHomeInterlock )
   END_RUNG
   RUNG wire#w1
      I_Contact( #AlwaysON )
      Coil( "ST10Cylinder".Cy[66].In.Error )
   END_RUNG
   // the same network as SCL:
   "ST10Cylinder".Cy[66].In.GoWorkInterlock := #AlwaysON AND #E_stop;
   "ST10Cylinder".Cy[66].In.GoHomeInterlock := #AlwaysON AND #E_stop;
   "ST10Cylinder".Cy[66].In.Error := #AlwaysON AND NOT #AlwaysON;
END_REGION

REGION Network 8: CY67 interface K-reserveLoadingStopperCylinder3_1
   RUNG wire#powerrail
      Contact( #AlwaysON )
      wire#w1
      Contact( #E_stop )
      wire#w2
      Coil( "ST10Cylinder".Cy[67].In.GoWorkInterlock )
   END_RUNG
   RUNG wire#w2
      Coil( "ST10Cylinder".Cy[67].In.GoHomeInterlock )
   END_RUNG
   RUNG wire#w1
      I_Contact( #AlwaysON )
      Coil( "ST10Cylinder".Cy[67].In.Error )
   END_RUNG
   // the same network as SCL:
   "ST10Cylinder".Cy[67].In.GoWorkInterlock := #AlwaysON AND #E_stop;
   "ST10Cylinder".Cy[67].In.GoHomeInterlock := #AlwaysON AND #E_stop;
   "ST10Cylinder".Cy[67].In.Error := #AlwaysON AND NOT #AlwaysON;
END_REGION

REGION Network 9: CY68 interface K-reserveLoadingStopperCylinder3_2
   RUNG wire#powerrail
      Contact( #AlwaysON )
      wire#w1
      Contact( #E_stop )
      wire#w2
      Coil( "ST10Cylinder".Cy[68].In.GoWorkInterlock )
   END_RUNG
   RUNG wire#w2
      Coil( "ST10Cylinder".Cy[68].In.GoHomeInterlock )
   END_RUNG
   RUNG wire#w1
      I_Contact( #AlwaysON )
      Coil( "ST10Cylinder".Cy[68].In.Error )
   END_RUNG
   // the same network as SCL:
   "ST10Cylinder".Cy[68].In.GoWorkInterlock := #AlwaysON AND #E_stop;
   "ST10Cylinder".Cy[68].In.GoHomeInterlock := #AlwaysON AND #E_stop;
   "ST10Cylinder".Cy[68].In.Error := #AlwaysON AND NOT #AlwaysON;
END_REGION

REGION Network 10: CY69 interface K-reserveLoadingStopperCylinder4_1
   RUNG wire#powerrail
      Contact( #AlwaysON )
      wire#w1
      Contact( #E_stop )
      wire#w2
      Coil( "ST10Cylinder".Cy[69].In.GoWorkInterlock )
   END_RUNG
   RUNG wire#w2
      Coil( "ST10Cylinder".Cy[69].In.GoHomeInterlock )
   END_RUNG
   RUNG wire#w1
      I_Contact( #AlwaysON )
      Coil( "ST10Cylinder".Cy[69].In.Error )
   END_RUNG
   // the same network as SCL:
   "ST10Cylinder".Cy[69].In.GoWorkInterlock := #AlwaysON AND #E_stop;
   "ST10Cylinder".Cy[69].In.GoHomeInterlock := #AlwaysON AND #E_stop;
   "ST10Cylinder".Cy[69].In.Error := #AlwaysON AND NOT #AlwaysON;
END_REGION

REGION Network 11: CY70 interface K-reserveLoadingStopperCylinder4_2
   RUNG wire#powerrail
      Contact( #AlwaysON )
      wire#w1
      Contact( #E_stop )
      wire#w2
      Coil( "ST10Cylinder".Cy[70].In.GoWorkInterlock )
   END_RUNG
   RUNG wire#w2
      Coil( "ST10Cylinder".Cy[70].In.GoHomeInterlock )
   END_RUNG
   RUNG wire#w1
      I_Contact( #AlwaysON )
      Coil( "ST10Cylinder".Cy[70].In.Error )
   END_RUNG
   // the same network as SCL:
   "ST10Cylinder".Cy[70].In.GoWorkInterlock := #AlwaysON AND #E_stop;
   "ST10Cylinder".Cy[70].In.GoHomeInterlock := #AlwaysON AND #E_stop;
   "ST10Cylinder".Cy[70].In.Error := #AlwaysON AND NOT #AlwaysON;
END_REGION
END_FUNCTION

FUNCTION "ST10Cyl_interface71-80" : Void   // FC1027, LAD
{ S7_Optimized_Access := 'FALSE' }
// stored: AutoNumber false, SetENOAutomatically false
   VAR_INPUT
      AlwaysON : Bool;
      E_stop : Bool;
   END_VAR
   VAR_TEMP
      tTest : Bool;
   END_VAR
BEGIN

REGION Network 1 (SCL): Cylinder 71-80 IO Interface (SCL)
   (*
   //Cylinder71 IO    K-reserveTakeStopperCylinder1_1
   //Input
   "ST10Cylinder".Cy[71].In.WorkPositionSensor := "oK-reserveTakeStopperCylinder1_1";
   "ST10Cylinder".Cy[71].In.HomePositionSensor := NOT "oK-reserveTakeStopperCylinder1_1";
   //Output
   "oK-reserveTakeStopperCylinder1_1" := "ST10Cylinder".Cy[71].Out.GoWorkPosition;
   #tTest := "ST10Cylinder".Cy[71].Out.GoHomePosition;

   //Cylinder72 IO    K-reserveTakeStopperCylinder1_2
   //Input
   "ST10Cylinder".Cy[72].In.WorkPositionSensor := "oK-reserveTakeStopperCylinder1_2";
   "ST10Cylinder".Cy[72].In.HomePositionSensor := NOT "oK-reserveTakeStopperCylinder1_2";
   //Output
   "oK-reserveTakeStopperCylinder1_2" := "ST10Cylinder".Cy[72].Out.GoWorkPosition;
   #tTest := "ST10Cylinder".Cy[72].Out.GoHomePosition;

   //Cylinder73 IO  K-reserveTakeStopperCylinder2_1
   //Input
   "ST10Cylinder".Cy[73].In.WorkPositionSensor := "oK-reserveTakeStopperCylinder2_1";
   "ST10Cylinder".Cy[73].In.HomePositionSensor := NOT "oK-reserveTakeStopperCylinder2_1";
   //Output
   "oK-reserveTakeStopperCylinder2_1" := "ST10Cylinder".Cy[73].Out.GoWorkPosition;
   #tTest := "ST10Cylinder".Cy[73].Out.GoHomePosition;

   //Cylinder74 IO  K-reserveTakeStopperCylinder2_2
   //Input
   "ST10Cylinder".Cy[74].In.WorkPositionSensor := "oK-reserveTakeStopperCylinder2_2";
   "ST10Cylinder".Cy[74].In.HomePositionSensor := NOT "oK-reserveTakeStopperCylinder2_2";
   //Output
   "oK-reserveTakeStopperCylinder2_2" := "ST10Cylinder".Cy[74].Out.GoWorkPosition;
   #tTest := "ST10Cylinder".Cy[74].Out.GoHomePosition;

   //Cylinder75 IO  K-reserveTakeStopperCylinder3_1
   //Input
   "ST10Cylinder".Cy[75].In.WorkPositionSensor := "oK-reserveTakeStopperCylinder3_1";
   "ST10Cylinder".Cy[75].In.HomePositionSensor := NOT "oK-reserveTakeStopperCylinder3_1";
   //Output
   "oK-reserveTakeStopperCylinder3_1" := "ST10Cylinder".Cy[75].Out.GoWorkPosition;
   #tTest := "ST10Cylinder".Cy[75].Out.GoHomePosition;

   //Cylinder76 IO  K-reserveTakeStopperCylinder3_2
   //Input
   "ST10Cylinder".Cy[76].In.WorkPositionSensor := "oK-reserveTakeStopperCylinder3_2";
   "ST10Cylinder".Cy[76].In.HomePositionSensor := NOT "oK-reserveTakeStopperCylinder3_2";
   //Output
   "oK-reserveTakeStopperCylinder3_2" := "ST10Cylinder".Cy[76].Out.GoWorkPosition;
   #tTest := "ST10Cylinder".Cy[76].Out.GoHomePosition;

   *)
END_REGION

REGION Network 2: CY71 interface K-reserveTakeStopperCylinder1_1
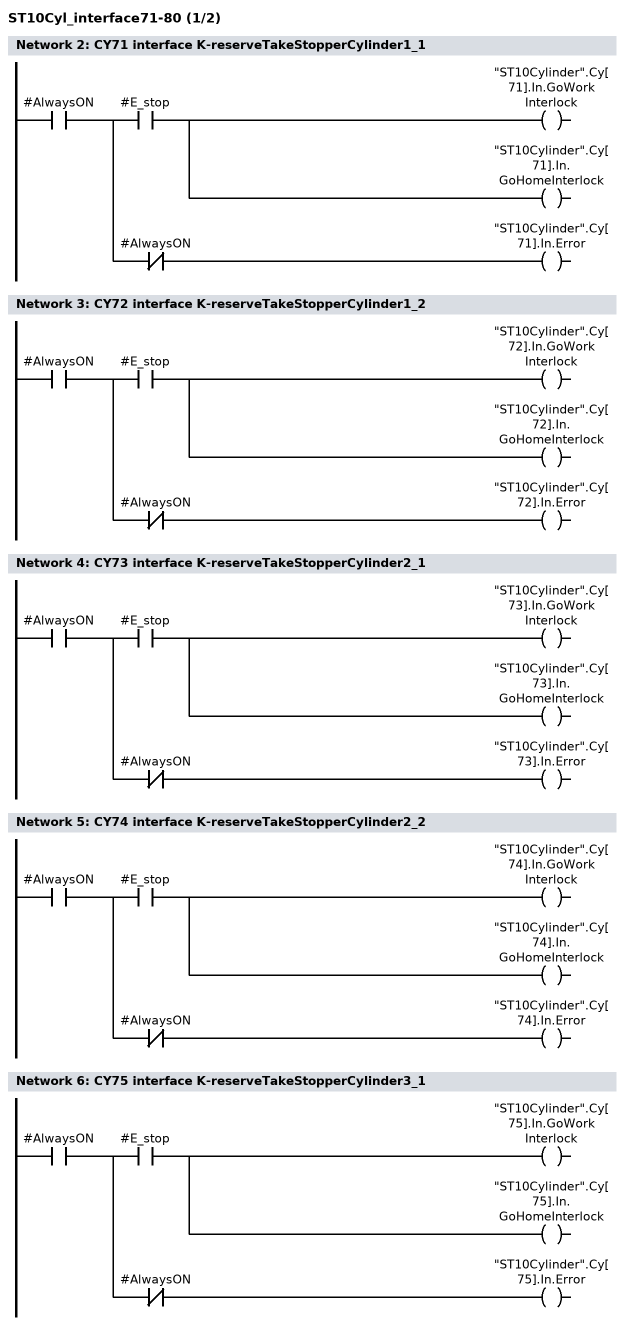
   RUNG wire#powerrail
      Contact( #AlwaysON )
      wire#w1
      Contact( #E_stop )
      wire#w2
      Coil( "ST10Cylinder".Cy[71].In.GoWorkInterlock )
   END_RUNG
   RUNG wire#w2
      Coil( "ST10Cylinder".Cy[71].In.GoHomeInterlock )
   END_RUNG
   RUNG wire#w1
      I_Contact( #AlwaysON )
      Coil( "ST10Cylinder".Cy[71].In.Error )
   END_RUNG
   // the same network as SCL:
   "ST10Cylinder".Cy[71].In.GoWorkInterlock := #AlwaysON AND #E_stop;
   "ST10Cylinder".Cy[71].In.GoHomeInterlock := #AlwaysON AND #E_stop;
   "ST10Cylinder".Cy[71].In.Error := #AlwaysON AND NOT #AlwaysON;
END_REGION

REGION Network 3: CY72 interface K-reserveTakeStopperCylinder1_2
   RUNG wire#powerrail
      Contact( #AlwaysON )
      wire#w1
      Contact( #E_stop )
      wire#w2
      Coil( "ST10Cylinder".Cy[72].In.GoWorkInterlock )
   END_RUNG
   RUNG wire#w2
      Coil( "ST10Cylinder".Cy[72].In.GoHomeInterlock )
   END_RUNG
   RUNG wire#w1
      I_Contact( #AlwaysON )
      Coil( "ST10Cylinder".Cy[72].In.Error )
   END_RUNG
   // the same network as SCL:
   "ST10Cylinder".Cy[72].In.GoWorkInterlock := #AlwaysON AND #E_stop;
   "ST10Cylinder".Cy[72].In.GoHomeInterlock := #AlwaysON AND #E_stop;
   "ST10Cylinder".Cy[72].In.Error := #AlwaysON AND NOT #AlwaysON;
END_REGION

REGION Network 4: CY73 interface K-reserveTakeStopperCylinder2_1
   RUNG wire#powerrail
      Contact( #AlwaysON )
      wire#w1
      Contact( #E_stop )
      wire#w2
      Coil( "ST10Cylinder".Cy[73].In.GoWorkInterlock )
   END_RUNG
   RUNG wire#w2
      Coil( "ST10Cylinder".Cy[73].In.GoHomeInterlock )
   END_RUNG
   RUNG wire#w1
      I_Contact( #AlwaysON )
      Coil( "ST10Cylinder".Cy[73].In.Error )
   END_RUNG
   // the same network as SCL:
   "ST10Cylinder".Cy[73].In.GoWorkInterlock := #AlwaysON AND #E_stop;
   "ST10Cylinder".Cy[73].In.GoHomeInterlock := #AlwaysON AND #E_stop;
   "ST10Cylinder".Cy[73].In.Error := #AlwaysON AND NOT #AlwaysON;
END_REGION

REGION Network 5: CY74 interface K-reserveTakeStopperCylinder2_2
   RUNG wire#powerrail
      Contact( #AlwaysON )
      wire#w1
      Contact( #E_stop )
      wire#w2
      Coil( "ST10Cylinder".Cy[74].In.GoWorkInterlock )
   END_RUNG
   RUNG wire#w2
      Coil( "ST10Cylinder".Cy[74].In.GoHomeInterlock )
   END_RUNG
   RUNG wire#w1
      I_Contact( #AlwaysON )
      Coil( "ST10Cylinder".Cy[74].In.Error )
   END_RUNG
   // the same network as SCL:
   "ST10Cylinder".Cy[74].In.GoWorkInterlock := #AlwaysON AND #E_stop;
   "ST10Cylinder".Cy[74].In.GoHomeInterlock := #AlwaysON AND #E_stop;
   "ST10Cylinder".Cy[74].In.Error := #AlwaysON AND NOT #AlwaysON;
END_REGION

